# B&R Automation Studio project NAELD004C00R10L518F00 (part 50)

#### Act_Link.st
```iecst
(** 2018-12-08 **)
ACTION Act_Link:

	//Machine --> AGV ---> Communication On & Machine itself RUN Mode
	IF p_bLinkOpsRun = TRUE THEN

		tyDTMagToAGV.bCI4Auto := TRUE;
	ELSE
		tyDTMagToAGV.bCI4Auto	:= FALSE;
	END_IF

	tyDTMagToAGV.bCI4Occupied 			:= p_bBufferMagPresent OR p_bMagConvLftSen OR p_bMagConvRgtSen ;

	fbMagEmptyTm(IN:= p_bMagConvLftSen = FALSE AND p_bBufferMagPresent = FALSE);
	IF p_bBufferMagPresent AND p_tyLinkBufferStat.bBffrMty THEN
		tyDTMagToAGV.bCI4MagazineEmpty		:=  TRUE;
	ELSIF fbMagEmptyTm.Q THEN
		tyDTMagToAGV.bCI4MagazineEmpty		:=  FALSE;
	END_IF

	IF p_bLinkAGVOnline THEN

		p_tyAGVToDTMag.bVEHAuto		:= p_tyLinkAGVtoDTMag.bVEHAuto;
		p_tyAGVToDTMag.bVEHInPos1	:= p_tyLinkAGVtoDTMag.bVEHInPos1;
		p_tyAGVToDTMag.bVEHInPos2 	:= p_tyLinkAGVtoDTMag.bVEHInPos2;
		p_tyAGVToDTMag.bVEHInPos3 	:= p_tyLinkAGVtoDTMag.bVEHInPos3;
		p_tyAGVToDTMag.bVEHInPos4 	:= p_tyLinkAGVtoDTMag.bVEHInPos4 AND bAGVInPosSen;
		p_tyAGVToDTMag.bVEH1Occupied	:= p_tyLinkAGVtoDTMag.bVEH1Occupied;
		p_tyAGVToDTMag.bVEH2Occupied	:= p_tyLinkAGVtoDTMag.bVEH2Occupied;
		p_tyAGVToDTMag.bVEH3Occupied	:= p_tyLinkAGVtoDTMag.bVEH3Occupied;
		p_tyAGVToDTMag.bVEH4Occupied	:= p_tyLinkAGVtoDTMag.bVEH4Occupied;
		p_tyAGVToDTMag.bVEHRunning	:= p_tyLinkAGVtoDTMag.bVEHRunning;

	ELSE

		p_tyAGVToDTMag.bVEHAuto		:= FALSE;
		p_tyAGVToDTMag.bVEHInPos1	:= FALSE;
		p_tyAGVToDTMag.bVEHInPos2 	:= FALSE;
		p_tyAGVToDTMag.bVEHInPos3 	:= FALSE;
		p_tyAGVToDTMag.bVEHInPos4 	:= FALSE;
		p_tyAGVToDTMag.bVEH1Occupied:= FALSE;
		p_tyAGVToDTMag.bVEH2Occupied:= FALSE;
		p_tyAGVToDTMag.bVEH3Occupied:= FALSE;
		p_tyAGVToDTMag.bVEH4Occupied:= FALSE;
		p_tyAGVToDTMag.bVEHRunning	:= FALSE;

	END_IF

	bAIVInPos := p_tyAGVToDTMag.bVEHInPos4;
	bAIVAuto := p_tyAGVToDTMag.bVEHAuto;
	bAIVOccupied := p_tyAGVToDTMag.bVEH4Occupied;
	bMagConvAuto := tyDTMagToAGV.bCI4Auto;
	bMagConvOccupied :=  tyDTMagToAGV.bCI4Occupied;

	tyDTMagToAGV.bCI4Running := bMagConvRun;
	tyDTMagToAGV.bCI4Rdy	:= bMagConvRdy;

	IF p_bNtParamAGVInPosSenPrep THEN
		fbInPosErrTimer(IN:= p_tyLinkAGVtoDTMag.bVEHInPos3 AND bAGVInPosSen = FALSE, PT:= T#10s);
		IF fbInPosErrTimer.Q THEN
			eStatus		:= Error;
			udiStatus	:= 10009;	//AIV Not In Position
		END_IF
	END_IF

	IF p_bNtParamAGVInPosSenPrep THEN
		bAGVInPosSen := p_bAGVInPosSen1 AND p_bAGVInPosSen2;
	ELSE
		bAGVInPosSen := TRUE;
	END_IF

END_ACTION
```

#### Act_Main.st
```iecst
(** 2019-01-20 **)
ACTION Act_Main:

	IF eStatOld <> eStat THEN

		fbTxInTimer(IN := FALSE);
		fbTxOutTimer(IN := FALSE);
		fbMagOutTrig(CLK := FALSE);

		bMcRunRdy				 	  := FALSE;
		bRdyEnt			 		   	  := FALSE;
		bRdyExit				  	  := FALSE;
		bMagConvRun    := FALSE;
		fbCheckErrorTim(IN:= FALSE);
		usiStep		:= 0;

		sStatTxt	:= a_sStatText[eStat];

		eStatOld	:= eStat;

		eStatus		:= Busy;
	END_IF

	//Main
	CASE eStat OF

		AGVMagActIdle:
			eStatus	:= Idle;
			bMagConvRdy := FALSE;

		AGVMagActEnter:

			IF eStatus = Idle OR eStatus = Busy THEN

				eStatus	:= Busy;
				bMagConvRdy := TRUE;

				IF usiStep = 0 THEN

					IF bAIVAuto AND bMagConvAuto
						OR p_bSOTAvailable
						THEN // ON Connection

						bMagConvRdy  := TRUE; //Allow VEH to Move In

						IF bAIVInPos OR p_bSOTRcvOk THEN // VEH is in Position to Enter

							bRdyEnt := TRUE;

						END_IF
					END_IF

					IF bRdyEnt THEN

						IF bAIVInPos OR p_bSOTRcvOk  THEN

							bMagConvRdy := FALSE; // Temporarily Not Allowed Other VEH while one VEH in Pos.

							IF p_bSOTErr THEN
								eStatus		:= Error;
								udiStatus	:= 10010;//SOT Sensor Error Has Been Activated;

							ELSIF (NOT bMagConvOccupied) (*AND p_tyAGVToDTMag.bVEHOccupied*) THEN

								bMcRunRdy	:= TRUE;

								bMagConvRun := TRUE;

								usiStep	:= 1;
							ELSE
								eStatus		:= Error;
								udiStatus	:= 10000;	//Magazine Is Present Before Entering
							END_IF

						ELSE
							eStatus		:= Error;
							udiStatus	:= 10001;	//AIV Not In Enter Position
						END_IF

					END_IF

				ELSIF usiStep = 1 THEN

					IF p_eDirection = ConvDirLToL OR p_eDirection = ConvDirLToR THEN
						bEndSen	:= p_bMagConvRgtSen;
					ELSE
						bEndSen	:= p_bMagConvLftSen;
					END_IF

					fbTxInTimer(IN := TRUE, PT := DINT_TO_TIME(p_diTxInTimeOut));

					IF bEndSen = TRUE (*AND p_tyAGVToDTMag.bVEHOccupied = FALSE*) THEN

						eStatus	:= Done;

						bMagConvRdy := TRUE; // Allow VEH to Move Out After Transfering Magazine

						bMagConvRun := FALSE;

					ELSIF fbTxInTimer.Q = TRUE THEN

						eStatus		:= Error;
						udiStatus	:= 10002;	//Transfer In Time Out While Transporting

					END_IF

					IF bAIVInPos = FALSE AND p_bSOTRcvOk = FALSE AND eStatus = Busy THEN

						eStatus		:= Error;
						udiStatus	:= 10001;	//AIV Not In Enter Position
					END_IF

					//					IF bAIVAuto = FALSE AND eStatus = Busy THEN
					//
					//						eStatus		:= Error;
					//						udiStatus	:= 10006;	//AIV Not In Enter Position
					//					END_IF
				END_IF

			END_IF

		AGVMagActExit:
			IF eStatus = Idle OR eStatus = Busy THEN

				eStatus	:= Busy;

				bMagConvRdy := TRUE;

				IF usiStep = 0 THEN

					IF bAIVAuto AND bMagConvAuto
						OR p_bSOTRdy
						THEN // ON Connection

						bMagConvRdy  := TRUE; //Allow VEH to Move In

						IF bAIVInPos OR p_bSOTRcvOk THEN // VEH is in Position to Exit

							bRdyExit := TRUE;

						END_IF
					END_IF

					IF bRdyExit THEN

						IF (bAIVInPos OR p_bSOTRcvOk) AND bAIVOccupied=FALSE THEN

							bMagConvRdy := FALSE; // Temporarily Not Allowed Other VEH while one VEH in Pos.

							IF bMagConvOccupied OR p_bSOTRdy = FALSE THEN

								bMcRunRdy	:= TRUE;

								bMagConvRun := TRUE;

								usiStep	:= 1;

							ELSE
								eStatus		:= Error;
								udiStatus	:= 10003;	//Magazine Is Not Present Before Exiting
							END_IF

						ELSE
							eStatus		:= Error;
							udiStatus	:= 10004;	//AIV Not In Exit Position
						END_IF
					END_IF

				ELSIF usiStep = 1 THEN

					IF p_bSOTErr THEN

						usiStep := 2;
					END_IF

					IF p_eDirection = ConvDirLToR OR p_eDirection = ConvDirRToR THEN
						bEndSen	:= p_bMagConvRgtSen;
					ELSE
						bEndSen	:= p_bMagConvLftSen;
					END_IF

					fbTxOutTimer(IN := TRUE, PT := DINT_TO_TIME(p_diTxOutTimeOut));

					IF bEndSen = FALSE AND (bAIVOccupied = TRUE OR p_bSOTRdy = FALSE) THEN

						usiStep := 2;

					ELSIF fbTxOutTimer.Q = TRUE THEN

						eStatus		:= Error;
						udiStatus	:= 10005;	//Transfer Out Time Out While Transporting

					END_IF

					IF bAIVInPos = FALSE AND p_bSOTRcvOk = FALSE AND eStatus = Busy THEN

						eStatus		:= Error;
						udiStatus	:= 10001;	//AIV Not In Enter Position
					END_IF

					//					IF bAIVAuto = FALSE AND eStatus = Busy THEN
					//
					//						eStatus		:= Error;
					//						udiStatus	:= 10006;	//AIV Not In Auto
					//					END_IF

				ELSIF usiStep = 2 THEN
					fbCheckErrorTim(IN:= TRUE);
					IF p_bSOTErr THEN
						eStatus		:= Error;
						udiStatus	:= 10010;	//SOT Error signal activated
					ELSIF fbCheckErrorTim.Q THEN
						usiStep := 3;
					END_IF

				ELSIF usiStep = 3 THEN
					bMagConvRdy 	   := TRUE; // Allow VEH to Move Out After Transfering Magazine

					bMagConvRun := FALSE;
					eStatus := Done;
				END_IF

			END_IF
	END_CASE

END_ACTION
```

#### Init.st
```iecst
(** 2019-01-20 **)
PROGRAM _INIT

	(* Always Change If Project Change *)

	sProgNm	:= 'AGVMag 4';

	//Physical Configuration

	//Pass Address To Global Address For External Use
	//Action, State & Status
	p_AGVMag4Stat		:= ADR(eStat);
	p_AGVMag4Status		:= ADR(eStatus);
	p_AGVMag4StatTxt	:= ADR(sStatTxt);

	//Alarm
	p_AGVMag4AlmData	:= ADR(tyAlmData);

	//Output
	p_AGVMag4RdyEnter		:= ADR(bRdyEnt);
	p_AGVMag4RdyExit		:= ADR(bRdyExit);
	p_AGVMag4McRunRdy		:= ADR(bMcRunRdy);
	p_AGVMag4DTMagToAGV		:= ADR(tyDTMagToAGV);

	(* Always Change If Project Change *)

END_PROGRAM
```

### Program Logical/SOT/USSOT1 (IEC) - 1.00.0 - NtSOT v5.00.0

#### Act_InitGlobal.st
```iecst
(** 2021-04-20 **)
ACTION Act_InitGlobal:

	(* Always Change If Project Change *)

	//Pass Data To Link
	p_bLinkOpsRun ACCESS p_OpsRun;
	p_bLinkSOTReadyOnFirst ACCESS p_NtParamSOTReadyOnFirst;

	//Pass Data To Internal Use
	p_udiRstErr ACCESS p_RstErrReset;
	p_bManual ACCESS p_UIMnlMod;
	p_diTransferInTO ACCESS p_McParamMag1ConvRunTmOut;
	p_bEn ACCESS p_McParamAGVComEn;
//	p_bVirtualEn ACCESS p_UIVSOTUSEn;
//	p_bUBAVirtual ACCESS p_UIVSOTUBA;
	p_tRstDlyTm ACCESS p_NtParamUSSOT1RstDlyTm;
	p_tSigInChkTm ACCESS p_NtParamUSSOT1SigInChkTm;
	p_sProgNm ACCESS p_NtParamUSSOT1ProgNm;
	p_bNtSettingsLoadDone ACCESS p_StartupNtSettingsLoadDone;

	(* Always Change If Project Change *)

END_ACTION
```

#### Act_Link.st
```iecst
(** 2021-04-20 **)
ACTION Act_Link:

	//Ready Receive
	IF p_bLinkSOTReadyOnFirst THEN
		p_bRdyRcv	:= TRUE;
	ELSE
		p_bRdyRcv ACCESS p_DISOT1Available;
	END_IF

	p_bLeftSen ACCESS p_DIMagConvEntSen1;
	p_bRightSen ACCESS p_DIMagPresentSen1;
	p_bUMA ACCESS p_DISOT1Available;
	p_bUMASize ACCESS p_DISOT1SizeLarge;
	p_bDirLToR := TRUE;

	p_bComplSigOn	:= p_bRightSen;

END_ACTION
```

#### Act_LinkAction.st
```iecst
(** 2021-04-20 **)
ACTION Act_LinkAction:

	IF p_bLinkOpsRun = TRUE THEN
		p_eAct ACCESS p_OpsMagConvLD1USSOTAct;
	ELSE
		p_eAct ACCESS ADR(eAct);
	END_IF

END_ACTION
```

### Program Logical/SOT/DSSOT1 (IEC) - 1.00.0 - NtSOT v5.00.0

#### Act_InitGlobal.st
```iecst
(** 2021-04-20 **)
ACTION Act_InitGlobal:

	(* Always Change If Project Change *)

	//Pass Data To Link
	p_bLinkOpsRun ACCESS p_OpsRun;

	//Pass Data To Internal Use
	p_udiRstErr ACCESS p_RstErrReset;
	p_bManual ACCESS p_UIMnlMod;
	p_diTransferOutTO ACCESS p_McParamMag1ConvRunTmOut;
	p_bEn ACCESS p_McParamAGVComEn;
//	p_bVirtualEn ACCESS p_UIVSOTDSEn;
//	p_bDSBVirtual ACCESS p_UIVSOTDSB;
	p_tRstDlyTm ACCESS p_NtParamDSSOT1RstDlyTm;
	p_tSigInChkTm ACCESS p_NtParamDSSOT1SigInChkTm;
	p_sProgNm ACCESS p_NtParamDSSOT1ProgNm;
	p_bNtSettingsLoadDone ACCESS p_StartupNtSettingsLoadDone;

	p_bMagSizeLarge ACCESS p_OpsMagConvLD1MagSizeL;

	(* Always Change If Project Change *)

END_ACTION
```

#### Act_Link.st
```iecst
(** 2021-04-20 **)
ACTION Act_Link:

	//Ready Send
	p_bRdySend	:= TRUE;

	p_bLeftSen ACCESS p_DIMagConvEntSen1;
	p_bRightSen ACCESS p_DIMagPresentSen1;
	p_bDSB ACCESS p_DISOT1Ready;

	//Send Complete Signal
	IF EDGENEG(p_bLeftSen) THEN
		p_bComplSigOn	:= TRUE;
	END_IF

	IF eStat <> SOTActRun THEN
		p_bComplSigOn	:= FALSE;
	END_IF

END_ACTION
```

#### Act_LinkAction.st
```iecst
(** 2021-04-20 **)
ACTION Act_LinkAction:

	IF p_bLinkOpsRun = TRUE THEN
		p_eAct ACCESS p_OpsMagConvLD1DSSOTAct;
	ELSE
		p_eAct ACCESS ADR(eAct);
	END_IF

END_ACTION
```

### Program Logical/SOT/USSOT2 (IEC) - 1.00.0 - NtSOT v5.00.0

#### Act_Alarm.st
```iecst
(** 2021-04-20 **)
ACTION Act_Alarm:

	//Error
	IF EDGEPOS(eStatus = Error) THEN

		tyAlmData.sProgNm		:= p_sProgNm;
		tyAlmData.udiCode		:= udiStatus;
		tyAlmData.eSeverity		:= AlmSeverityError;
		tyAlmData.udiRunTime	:= tyAlmData.udiRunTime + 1;
		tyAlmData.bAlm			:= TRUE;
		tyAlmData.udiModuleNum  := udiModuleNum;
		g_sUSSOTProgNm		:= p_sProgNm;
		//Get Error Message
		IF tyAlmData.udiCode < 10000 OR tyAlmData.udiCode > 10099 THEN
			tyAlmData.sAlmMsg	:= 'Unknown';
			tyAlmData.sRcyMsg	:= 'Unknown';
		ELSE
			tyAlmData.sAlmMsg	:= a_tyAlmText[tyAlmData.udiCode].sAlmText;
			tyAlmData.sRcyMsg	:= a_tyAlmText[tyAlmData.udiCode].sRcyText;
		END_IF

		sStatTxt	:= tyAlmData.sAlmMsg;

	ELSIF bRstErr AND (tyAlmData.udiCode <> 0) THEN

		tyAlmData.udiCode	:= 0;
		tyAlmData.eSeverity	:= AlmSeverityNA;
		tyAlmData.sAlmMsg	:= '';
		tyAlmData.sRcyMsg	:= '';
		tyAlmData.bAlm			:= FALSE;
		sStatTxt	:= a_sStatText[eStat];

	END_IF

END_ACTION
```

#### Act_InitGlobal.st
```iecst
(** 2021-04-20 **)
ACTION Act_InitGlobal:

	(* Always Change If Project Change *)

	//Pass Data To Link
	p_bLinkOpsRun ACCESS p_OpsRun;
	p_bLinkSOTReadyOnFirst ACCESS p_NtParamSOTReadyOnFirst;

	//Pass Data To Internal Use
	p_udiRstErr ACCESS p_RstErrReset;
	p_bManual ACCESS p_UIMnlMod;
	p_diTransferInTO ACCESS p_McParamMag2ConvRunTmOut;
	p_bEn ACCESS p_McParamAGVComEn;
//	p_bVirtualEn ACCESS p_UIVSOTUSEn;
//	p_bUBAVirtual ACCESS p_UIVSOTUBA;
	p_tRstDlyTm ACCESS p_NtParamUSSOT2RstDlyTm;
	p_tSigInChkTm ACCESS p_NtParamUSSOT2SigInChkTm;
	p_sProgNm ACCESS p_NtParamUSSOT2ProgNm;
	p_bNtSettingsLoadDone ACCESS p_StartupNtSettingsLoadDone;

	(* Always Change If Project Change *)

END_ACTION
```

#### Act_Link.st
```iecst
(** 2021-04-20 **)
ACTION Act_Link:

	//Ready Receive
	IF p_bLinkSOTReadyOnFirst THEN
		p_bRdyRcv	:= TRUE;
	ELSE
		p_bRdyRcv ACCESS p_DISOT2Available;
	END_IF

	p_bLeftSen ACCESS p_DIMagConvEntSen2;
	p_bRightSen ACCESS p_DIMagPresentSen2;
	p_bUMA ACCESS p_DISOT2Available;
	p_bUMASize ACCESS p_DISOT2SizeLarge;
	p_bDirLToR := TRUE;

	p_bComplSigOn	:= p_bRightSen;

END_ACTION
```

#### Act_LinkAction.st
```iecst
(** 2021-04-20 **)
ACTION Act_LinkAction:

	IF p_bLinkOpsRun = TRUE THEN
		p_eAct ACCESS p_OpsMagConvLD2USSOTAct;
	ELSE
		p_eAct ACCESS ADR(eAct);
	END_IF

END_ACTION
```

### Program Logical/SOT/DSSOT2 (IEC) - 1.00.0 - NtSOT v5.00.0

#### Act_InitGlobal.st
```iecst
(** 2021-04-20 **)
ACTION Act_InitGlobal:

	(* Always Change If Project Change *)

	//Pass Data To Link
	p_bLinkOpsRun ACCESS p_OpsRun;

	//Pass Data To Internal Use
	p_udiRstErr ACCESS p_RstErrReset;
	p_bManual ACCESS p_UIMnlMod;
	p_diTransferOutTO ACCESS p_McParamMag2ConvRunTmOut;
	p_bEn ACCESS p_McParamAGVComEn;
//	p_bVirtualEn ACCESS p_UIVSOTDSEn;
//	p_bDSBVirtual ACCESS p_UIVSOTDSB;
	p_tRstDlyTm ACCESS p_NtParamDSSOT2RstDlyTm;
	p_tSigInChkTm ACCESS p_NtParamDSSOT2SigInChkTm;
	p_sProgNm ACCESS p_NtParamDSSOT2ProgNm;
	p_bNtSettingsLoadDone ACCESS p_StartupNtSettingsLoadDone;

	p_bMagSizeLarge ACCESS p_OpsMagConvLD2MagSizeL;

	(* Always Change If Project Change *)

END_ACTION
```

#### Act_Link.st
```iecst
(** 2021-04-20 **)
ACTION Act_Link:

	//Ready Send
	p_bRdySend	:= TRUE;

	p_bLeftSen ACCESS p_DIMagConvEntSen2;
	p_bRightSen ACCESS p_DIMagPresentSen2;
	p_bDSB ACCESS p_DISOT2Ready;

	//Send Complete Signal
	IF EDGENEG(p_bLeftSen) THEN
		p_bComplSigOn	:= TRUE;
	END_IF

	IF eStat <> SOTActRun THEN
		p_bComplSigOn	:= FALSE;
	END_IF

END_ACTION
```

#### Act_LinkAction.st
```iecst
(** 2021-04-20 **)
ACTION Act_LinkAction:

	IF p_bLinkOpsRun = TRUE THEN
		p_eAct ACCESS p_OpsMagConvLD2DSSOTAct;
	ELSE
		p_eAct ACCESS ADR(eAct);
	END_IF

END_ACTION
```

### USSOT3.var - Change By Project
```iecst
(*2021-03-19*)
(**)
(*Action & State & Status*)
VAR
	p_USSOT3Stat : UDINT;
	p_USSOT3Status : UDINT;
	p_USSOT3StatTxt : UDINT;
END_VAR
(**)
(*Alarm*)
VAR
	p_USSOT3AlmData : UDINT;
END_VAR
(**)
(*Output*)
VAR
	p_USSOT3USRdy : UDINT;
	p_USSOT3USLargeMagRdy : UDINT;
	p_USSOT3DSRdy : UDINT;
	p_USSOT3Transporting : UDINT;
	p_USSOT3ConvStart : UDINT;
	p_USSOT3ConvStop : UDINT;
	p_USSOT3USB : UDINT;
	p_USSOT3Virtual : UDINT;
END_VAR
```

### Program Logical/SOT/USSOT3 (IEC) - 1.00.0 - NtSOT v5.00.0

#### Act_InitGlobal.st
```iecst
(** 2021-04-20 **)
ACTION Act_InitGlobal:

	(* Always Change If Project Change *)

	//Pass Data To Link
	p_bLinkOpsRun ACCESS p_OpsRun;
	p_bLinkSOTReadyOnFirst ACCESS p_NtParamSOTReadyOnFirst;

	//Pass Data To Internal Use
	p_udiRstErr ACCESS p_RstErrReset;
	p_bManual ACCESS p_UIMnlMod;
	p_diTransferInTO ACCESS p_McParamMag3ConvRunTmOut;
	p_bEn ACCESS p_McParamAGVComEn;
//	p_bVirtualEn ACCESS p_UIVSOTUSEn;
//	p_bUBAVirtual ACCESS p_UIVSOTUBA;
	p_tRstDlyTm ACCESS p_NtParamUSSOT3RstDlyTm;
	p_tSigInChkTm ACCESS p_NtParamUSSOT3SigInChkTm;
	p_sProgNm ACCESS p_NtParamUSSOT3ProgNm;
	p_bNtSettingsLoadDone ACCESS p_StartupNtSettingsLoadDone;

	(* Always Change If Project Change *)

END_ACTION
```

#### Act_LinkAction.st
```iecst
(** 2021-04-20 **)
ACTION Act_LinkAction:

	IF p_bLinkOpsRun = TRUE THEN
		p_eAct ACCESS p_OpsMagConvLD3USSOTAct;
	ELSE
		p_eAct ACCESS ADR(eAct);
	END_IF

END_ACTION
```

### Program Logical/SOT/DSSOT3 (IEC) - 1.00.0 - NtSOT v5.00.0

#### Act_InitGlobal.st
```iecst
(** 2021-04-20 **)
ACTION Act_InitGlobal:

	(* Always Change If Project Change *)

	//Pass Data To Link
	p_bLinkOpsRun ACCESS p_OpsRun;

	//Pass Data To Internal Use
	p_udiRstErr ACCESS p_RstErrReset;
	p_bManual ACCESS p_UIMnlMod;
	p_diTransferOutTO ACCESS p_McParamMag3ConvRunTmOut;
	p_bEn ACCESS p_McParamAGVComEn;
//	p_bVirtualEn ACCESS p_UIVSOTDSEn;
//	p_bDSBVirtual ACCESS p_UIVSOTDSB;
	p_tRstDlyTm ACCESS p_NtParamDSSOT3RstDlyTm;
	p_tSigInChkTm ACCESS p_NtParamDSSOT3SigInChkTm;
	p_sProgNm ACCESS p_NtParamDSSOT3ProgNm;
	p_bNtSettingsLoadDone ACCESS p_StartupNtSettingsLoadDone;

	p_bMagSizeLarge ACCESS p_OpsMagConvLD3MagSizeL;

	(* Always Change If Project Change *)

END_ACTION
```

#### Act_LinkAction.st
```iecst
(** 2021-04-20 **)
ACTION Act_LinkAction:

	IF p_bLinkOpsRun = TRUE THEN
		p_eAct ACCESS p_OpsMagConvLD3DSSOTAct;
	ELSE
		p_eAct ACCESS ADR(eAct);
	END_IF

END_ACTION
```

### USSOT4.var - Change By Project
```iecst
(*2021-04-19*)
(**)
(*Action & State & Status*)
VAR
	p_USSOT4Stat : UDINT;
	p_USSOT4Status : UDINT;
	p_USSOT4StatTxt : UDINT;
END_VAR
(**)
(*Alarm*)
VAR
	p_USSOT4AlmData : UDINT;
END_VAR
(**)
(*Output*)
VAR
	p_USSOT4USRdy : UDINT;
	p_USSOT4USLargeMagRdy : UDINT;
	p_USSOT4DSRdy : UDINT;
	p_USSOT4Transporting : UDINT;
	p_USSOT4ConvStart : UDINT;
	p_USSOT4ConvStop : UDINT;
	p_USSOT4USB : UDINT;
	p_USSOT4Virtual : UDINT;
END_VAR
```

### Program Logical/SOT/USSOT4 (IEC) - 1.00.0 - NtSOT v5.00.0

#### InputRef_Link.var
```iecst
(*2021-04-20*)
(**)
VAR
	p_bLinkOpsRun : REFERENCE TO BOOL;
	p_bLinkSOTReadyOnFirst : REFERENCE TO BOOL;
END_VAR
```

#### Act_InitGlobal.st
```iecst
(** 2021-04-20 **)
ACTION Act_InitGlobal:

	(* Always Change If Project Change *)

	//Pass Data To Link
	p_bLinkOpsRun ACCESS p_OpsRun;
	p_bLinkSOTReadyOnFirst ACCESS p_NtParamSOTReadyOnFirst;

	//Pass Data To Internal Use
	p_udiRstErr ACCESS p_RstErrReset;
	p_bManual ACCESS p_UIMnlMod;
	p_diTransferInTO ACCESS p_McParamMag4ConvRunTmOut;
	p_bEn ACCESS p_McParamAGVComEn;
//	p_bVirtualEn ACCESS p_UIVSOTUSEn;
//	p_bUBAVirtual ACCESS p_UIVSOTUBA;
	p_tRstDlyTm ACCESS p_NtParamUSSOT4RstDlyTm;
	p_tSigInChkTm ACCESS p_NtParamUSSOT4SigInChkTm;
	p_sProgNm ACCESS p_NtParamUSSOT4ProgNm;
	p_bNtSettingsLoadDone ACCESS p_StartupNtSettingsLoadDone;

	(* Always Change If Project Change *)

END_ACTION
```

#### Act_Link.st
```iecst
(** 2021-04-20 **)
ACTION Act_Link:

	//Ready Receive
	IF p_bLinkSOTReadyOnFirst THEN
		p_bRdyRcv	:= TRUE;
	ELSE
		p_bRdyRcv ACCESS p_DISOT4Available;
	END_IF
	p_bLeftSen ACCESS p_DIMagConvEntSen4;
	p_bRightSen ACCESS p_DIMagPresentSen4;
	p_bUMA ACCESS p_DISOT4Available;
	p_bUMASize ACCESS p_DISOT4SizeLarge;
	p_bDirLToR := TRUE;

	p_bComplSigOn	:= p_bRightSen;

END_ACTION
```

#### Act_LinkAction.st
```iecst
(** 2021-04-20 **)
ACTION Act_LinkAction:

	IF p_bLinkOpsRun = TRUE THEN
		p_eAct ACCESS p_OpsMagConvLD4USSOTAct;
	ELSE
		p_eAct ACCESS ADR(eAct);
	END_IF

END_ACTION
```

#### Init.st
```iecst
(** 2021-04-20 **)
PROGRAM _INIT

	(* Always Change If Project Change *)

	//Pass Address To Global Address For External Use
	//Action, State & Status
	p_USSOT4Stat		:= ADR(eStat);
	p_USSOT4Status	:= ADR(eStatus);
	p_USSOT4StatTxt	:= ADR(sStatTxt);

	//Alarm
	p_USSOT4AlmData	:= ADR(tyAlmData);

	//Output
	p_USSOT4USRdy			:= ADR(bUSRdy);
	p_USSOT4USLargeMagRdy	:= ADR(bUSLargeMagRdy);
	p_USSOT4DSRdy			:= ADR(bDSRdy);
	p_USSOT4Transporting	:= ADR(bTransporting);
	p_USSOT4ConvStart		:= ADR(bConvStart);
	p_USSOT4ConvStop		:= ADR(bConvStop);
	p_USSOT4USB				:= ADR(bUSB);
	p_USSOT4Virtual			:= ADR(bVirtual);

	(* Always Change If Project Change *)

END_PROGRAM
```

### DSSOT4.var - Change By Project
```iecst
(*2021-04-20*)
(**)
(*Action & State & Status*)
VAR
	p_DSSOT4Stat : UDINT;
	p_DSSOT4Status : UDINT;
	p_DSSOT4StatTxt : UDINT;
END_VAR
(**)
(*Alarm*)
VAR
	p_DSSOT4AlmData : UDINT;
END_VAR
(**)
(*Output*)
VAR
	p_DSSOT4USRdy : UDINT;
	p_DSSOT4DSRdy : UDINT;
	p_DSSOT4Transporting : UDINT;
	p_DSSOT4ConvStart : UDINT;
	p_DSSOT4ConvStop : UDINT;
	p_DSSOT4DBA : UDINT;
	p_DSSOT4MagSizeLarge : UDINT;
	p_DSSOT4Virtual : UDINT;
END_VAR
```

### Program Logical/SOT/DSSOT4 (IEC) - 1.00.0 - NtSOT v5.00.0

#### Act_InitGlobal.st
```iecst
(** 2021-04-20 **)
ACTION Act_InitGlobal:

	(* Always Change If Project Change *)

	//Pass Data To Link
	p_bLinkOpsRun ACCESS p_OpsRun;

	//Pass Data To Internal Use
	p_udiRstErr ACCESS p_RstErrReset;
	p_bManual ACCESS p_UIMnlMod;
	p_diTransferOutTO ACCESS p_McParamMag4ConvRunTmOut;
	p_bEn ACCESS p_McParamAGVComEn;
//	p_bVirtualEn ACCESS p_UIVSOTDSEn;
//	p_bDSBVirtual ACCESS p_UIVSOTDSB;
	p_tRstDlyTm ACCESS p_NtParamDSSOT4RstDlyTm;
	p_tSigInChkTm ACCESS p_NtParamDSSOT4SigInChkTm;
	p_sProgNm ACCESS p_NtParamDSSOT4ProgNm;
	p_bNtSettingsLoadDone ACCESS p_StartupNtSettingsLoadDone;

	p_bMagSizeLarge ACCESS p_OpsMagConvLD4MagSizeL;

	(* Always Change If Project Change *)

END_ACTION
```

#### Act_Link.st
```iecst
(** 2021-04-20 **)
ACTION Act_Link:

	//Ready Send
	p_bRdySend	:= TRUE;

	p_bLeftSen ACCESS p_DIMagConvEntSen4;
	p_bRightSen ACCESS p_DIMagPresentSen4;
	p_bDSB ACCESS p_DISOT4Ready;

	//Send Complete Signal
	IF EDGENEG(p_bLeftSen) THEN
		p_bComplSigOn	:= TRUE;
	END_IF

	IF eStat <> SOTActRun THEN
		p_bComplSigOn	:= FALSE;
	END_IF

END_ACTION
```

#### Act_LinkAction.st
```iecst
(** 2021-04-20 **)
ACTION Act_LinkAction:

	IF p_bLinkOpsRun = TRUE THEN
		p_eAct ACCESS p_OpsMagConvLD4DSSOTAct;
	ELSE
		p_eAct ACCESS ADR(eAct);
	END_IF

END_ACTION
```

#### Init.st
```iecst
(** 2021-04-20 **)
PROGRAM _INIT

	(* Always Change If Project Change *)

	//Pass Address To Global Address For External Use
	//Action, State & Status
	p_DSSOT4Stat		:= ADR(eStat);
	p_DSSOT4Status		:= ADR(eStatus);
	p_DSSOT4StatTxt		:= ADR(sStatTxt);

	//Alarm
	p_DSSOT4AlmData	:= ADR(tyAlmData);

	//Output
	p_DSSOT4USRdy			:= ADR(bUSRdy);
	p_DSSOT4DSRdy			:= ADR(bDSRdy);
	p_DSSOT4Transporting	:= ADR(bTransporting);
	p_DSSOT4ConvStart		:= ADR(bConvStart);
	p_DSSOT4ConvStop		:= ADR(bConvStop);
	p_DSSOT4DBA				:= ADR(bDBA);
	p_DSSOT4Virtual			:= ADR(bVirtual);
	p_DSSOT4MagSizeLarge	:= ADR(bDSMagSizeLarge);

	(* Always Change If Project Change *)

END_PROGRAM
```

### Program Logical/Machine/Machine (IEC) - 1.00.0 - 

#### InputRef.var
```iecst
(*2019-03-22*)
(**)
(*General*)
VAR
	p_udiRstErr : REFERENCE TO UDINT;
END_VAR
(**)
(*Configuration*)
VAR
	p_bOpsRun : REFERENCE TO BOOL;
	p_bDIPressureSW : REFERENCE TO BOOL;
	p_diProdRcpCurrRcpWidth : REFERENCE TO DINT;
	p_diMagRcpCurrRcpMaxWidth : REFERENCE TO DINT;
	p_eStartupStep : REFERENCE TO eStartupStep;
END_VAR
(**)
VAR
	p_sProgNm : REFERENCE TO STRING[15];
	p_bNtSettingsLoadDone : REFERENCE TO BOOL;
	p_eLinkMag : REFERENCE TO eLDMag;
	p_usiLinkMod : REFERENCE TO USINT;
	p_bMcParamHermesSvyEn : REFERENCE TO BOOL;
END_VAR
```

#### Local.var
```iecst
(*2019-03-25*)
(**)
(*Local Action, State & Status*)
VAR
	eStatus : eFBStatus := Idle;
	udiStatus : UDINT := 0;
	udiStatus1 : UDINT := 0;
END_VAR
(**)
(*Local Alarm*)
VAR
	tyAlmData : tyAlmDat;
	tyAlmData1 : tyAlmDat;
	a_tyAlmText : ARRAY[10000..10099] OF tyAlmTxt := [(sAlmText:='Selected Product Width Exceeds Selected Magazine Maximum Board Width',sRcyText:='Please Reselect  Product or Magazine '),99(0)];
END_VAR
(**)
(*Local Output*)
(**)
(*Local Input*)
VAR
	udiRstErr : UDINT := 0;
END_VAR
(**)
VAR
	bOpsRun : BOOL;
	diProdRcpCurrRcpWidth : DINT;
	diMagRcpCurrRcpMaxWidth : DINT;
END_VAR
(**)
VAR
	sProgNm : STRING[15] := 'Machine';
	bNtSettingsLoadDone : BOOL := TRUE;
END_VAR
(**)
(*Local*)
VAR
	bRstErr : BOOL;
	udiRstErrOld : UDINT;
	bInitDone : BOOL;
	bInitialDone : BOOL;
END_VAR
(**)
VAR
	sBarcodeOut : STRING[255];
	bUSBDisconnected : BOOL;
	eStat : eUSBRdrAction := USBRdrActIdle;
	eMainStatus : eFBStatus := Idle;
	sStatTxt : STRING[200] := '';
	udiModuleNum : UDINT := 5951;
END_VAR
```

#### Act_Alarm.st
```iecst
(** 2019-03-25 **)
ACTION Act_Alarm:

	//Error
	IF EDGEPOS(eStatus = Error) THEN

		tyAlmData.sProgNm		:= p_sProgNm;
		tyAlmData.udiCode		:= udiStatus;
		tyAlmData.eSeverity		:= AlmSeverityError;
		tyAlmData.udiRunTime	:= tyAlmData.udiRunTime + 1;
		tyAlmData.bAlm			:= TRUE;
		tyAlmData.udiModuleNum  := udiModuleNum;
		g_sMachineProgNm		:= p_sProgNm;
		//Get Error Message
		IF tyAlmData.udiCode < 10000 OR tyAlmData.udiCode > 10099 THEN
			tyAlmData.sAlmMsg	:= 'Unknown';
			tyAlmData.sRcyMsg	:= 'Unknown';
		ELSE
			tyAlmData.sAlmMsg	:= a_tyAlmText[tyAlmData.udiCode].sAlmText;
			tyAlmData.sRcyMsg	:= a_tyAlmText[tyAlmData.udiCode].sRcyText;
		END_IF

	END_IF

END_ACTION
```

#### Act_Background.st
```iecst
(** 2019-01-23 **)
ACTION Act_Background:

	IF (p_diProdRcpCurrRcpWidth > p_diMagRcpCurrRcpMaxWidth) AND (eStatus <> Error) AND p_bMcParamHermesSvyEn =FALSE THEN

		eStatus		:= Error;
		udiStatus   := 10000;

	END_IF

	//Reset Error
	IF (eStatus = Error) AND bRstErr THEN
		eStatus		:= Idle;
		udiStatus	:= 0;
	END_IF

END_ACTION
```

#### Act_InitGlobal.st
```iecst
(** 2019-04-09 **)
ACTION Act_InitGlobal:

	(* Always Change If Project Change *)

	//Pass Data To Link
	p_eLinkMag ACCESS p_NtParamProjMag;
	p_usiLinkMod ACCESS p_ProdRcpCurrRcp0McMod;
	p_bMcParamHermesSvyEn ACCESS p_McParamHermesSvyEn;

	//Pass Data To Internal Use
	p_udiRstErr ACCESS p_RstErrReset;

	p_bOpsRun ACCESS p_OpsRun;
	p_eStartupStep ACCESS p_StartupStep;

	p_sProgNm ACCESS p_NtParamMcProgNm;
	p_bNtSettingsLoadDone ACCESS p_StartupNtSettingsLoadDone;

	(* Always Change If Project Change *)

END_ACTION
```

#### Act_Initial.st
```iecst
(** 2018-12-07 **)
ACTION Act_Initial:

	//Initial

END_ACTION
```

#### Act_Link.st
```iecst
(** 2018-12-11 **)
ACTION Act_Link:

	IF p_eLinkMag = LDMagQuadruple THEN
		CASE p_usiLinkMod OF
			0,2:
				p_diProdRcpCurrRcpWidth ACCESS p_ProdRcpCurrRcp0Width;
				p_diMagRcpCurrRcpMaxWidth ACCESS p_MagRcpCurrRcpMagMaxBrdWidth;

			1:
				p_diProdRcpCurrRcpWidth ACCESS p_ProdRcpCurrRcp0WidthRear;
				p_diMagRcpCurrRcpMaxWidth ACCESS p_MagRcpCurrRcpMagMaxBrdWidth1;
		END_CASE
	ELSE
		p_diProdRcpCurrRcpWidth ACCESS p_ProdRcpCurrRcp0Width;
		p_diMagRcpCurrRcpMaxWidth ACCESS p_MagRcpCurrRcpMagMaxBrdWidth;
	END_IF

END_ACTION
```

#### Init.st
```iecst
(** 2019-03-22 **)
PROGRAM _INIT

	(* Always Change If Project Change *)

	//Pass Address To Global Address For External Use
	//Action, State & Status

	//Alarm
	p_McAlmData		:= ADR(tyAlmData);
	p_McInfoData1	:= ADR(tyAlmData1);

	//Output

END_PROGRAM
```

### Machine1.var - Change By Project
```iecst
(*2018-12-07*)
(**)
(*Action & State & Status*)
(**)
(*Alarm*)
VAR
	p_Mc1AlmData : UDINT;
	p_Mc1InfoData1 : UDINT;
END_VAR
(**)
(*Output*)
```

### Program Logical/Machine/Machine1 (IEC, version 1.00.0) - 1.00.0 - 

#### Init.st - Change By Project
```iecst
(** 2019-03-22 **)
PROGRAM _INIT

	(* Always Change If Project Change *)

	//Pass Address To Global Address For External Use
	//Action, State & Status

	//Alarm
	p_Mc1AlmData		:= ADR(tyAlmData);
	p_Mc1InfoData1		:= ADR(tyAlmData1);

	//Output

	(* Always Change If Project Change *)

END_PROGRAM
```

#### Act_InitGlobal.st - Change By Project
```iecst
(** 2019-04-09 **)
ACTION Act_InitGlobal:

	(* Always Change If Project Change *)

	//Pass Data To Link
	p_eLinkMag ACCESS p_NtParamProjMag;
	p_usiLinkMod ACCESS p_ProdRcpCurrRcp0McMod;
	//Pass Data To Internal Use
	p_udiRstErr ACCESS p_RstErrReset;

	p_bOpsRun ACCESS p_OpsRun;
	p_eStartupStep ACCESS p_StartupStep;

	p_sProgNm ACCESS p_NtParamMc1ProgNm;
	p_bNtSettingsLoadDone ACCESS p_StartupNtSettingsLoadDone;

	(* Always Change If Project Change *)

END_ACTION
```

#### Act_Link.st - Change By Project
```iecst
(** 2018-12-11 **)
ACTION Act_Link:

	IF p_eLinkMag = LDMagQuadruple THEN
		CASE p_usiLinkMod OF
			1,2:
				p_diProdRcpCurrRcpWidth ACCESS p_ProdRcpCurrRcp0WidthRear;
				p_diMagRcpCurrRcpMaxWidth ACCESS p_MagRcpCurrRcpMagMaxBrdWidth1;

			0:
				p_diProdRcpCurrRcpWidth ACCESS p_ProdRcpCurrRcp0Width;
				p_diMagRcpCurrRcpMaxWidth ACCESS p_MagRcpCurrRcpMagMaxBrdWidth;
		END_CASE
	ELSE
		p_diProdRcpCurrRcpWidth := 0;
		p_diMagRcpCurrRcpMaxWidth := p_NtParamProdRcpMaxWidth;
	END_IF

END_ACTION
```

#### Cyclic.st - Change By Project
```iecst
(** 2019-03-22 **)
PROGRAM _CYCLIC

	IF bInitDone = FALSE THEN
		bInitDone	:= TRUE;

		Act_InitLocal;
		Act_InitGlobal;

	ELSIF bInitialDone = FALSE THEN

		//Special Case --> only after reading Current Recipe --> Excusively for Machine with Magazine Maximum Board Width Setting

		IF p_bNtSettingsLoadDone = TRUE AND p_eStartupStep = StartupStepUsrMgmt  THEN
			bInitialDone	:= TRUE;

			Act_Initial;
		END_IF

	ELSE

		Act_RstErr;
		Act_Link;
		Act_Background;
		Act_Alarm;
		Act_AlarmInfo1;

	END_IF

END_PROGRAM
```

#### Act_Alarm.st - Change By Project
```iecst
(** 2019-03-25 **)
ACTION Act_Alarm:

	//Error
	IF EDGEPOS(eStatus = Error) THEN

		tyAlmData.sProgNm		:= p_sProgNm;
		tyAlmData.udiCode		:= udiStatus;
		tyAlmData.eSeverity		:= AlmSeverityError;
		tyAlmData.udiRunTime	:= tyAlmData.udiRunTime + 1;
		tyAlmData.bAlm			:= TRUE;
		tyAlmData.udiModuleNum  := udiModuleNum;
		g_sMachineProgNm		:= p_sProgNm;
		//Get Error Message
		IF tyAlmData.udiCode < 10000 OR tyAlmData.udiCode > 10099 THEN
			tyAlmData.sAlmMsg	:= 'Unknown';
			tyAlmData.sRcyMsg	:= 'Unknown';
		ELSE
			tyAlmData.sAlmMsg	:= a_tyAlmText[tyAlmData.udiCode].sAlmText;
			tyAlmData.sRcyMsg	:= a_tyAlmText[tyAlmData.udiCode].sRcyText;
		END_IF

	END_IF

END_ACTION
```

#### InputRef.var - Change By Project
```iecst
(*2019-03-22*)
(**)
(*General*)
VAR
	p_udiRstErr : REFERENCE TO UDINT;
	p_bPrep : REFERENCE TO BOOL;
	p_bEn : REFERENCE TO BOOL;
	p_bDis : REFERENCE TO BOOL;
END_VAR
(**)
(*Configuration*)
VAR
	p_bOpsRun : REFERENCE TO BOOL;
	p_bDIPressureSW : REFERENCE TO BOOL;
	p_diProdRcpCurrRcpWidth : REFERENCE TO DINT;
	p_diMagRcpCurrRcpMaxWidth : REFERENCE TO DINT;
	p_eStartupStep : REFERENCE TO eStartupStep;
END_VAR
(**)
VAR
	p_sProgNm : REFERENCE TO STRING[15];
	p_bNtSettingsLoadDone : REFERENCE TO BOOL;
	p_eLinkMag : REFERENCE TO eLDMag;
	p_usiLinkMod : REFERENCE TO USINT;
END_VAR
```

#### Local.var - Change By Project
```iecst
(*2019-03-25*)
(**)
(*Local Action, State & Status*)
VAR
	eStatus : eFBStatus := Idle;
	udiStatus : UDINT := 0;
	udiStatus1 : UDINT := 0;
END_VAR
(**)
(*Local Alarm*)
VAR
	tyAlmData : tyAlmDat;
	tyAlmData1 : tyAlmDat;
	a_tyAlmText : ARRAY[10000..10099] OF tyAlmTxt := [(sAlmText:='Selected Product Width Exceeds Slected Magazine Maximum Board Width',sRcyText:='Please Reslect  Product or Magazine '),99((0))];
END_VAR
(**)
(*Local Output*)
(**)
(*Local Input*)
VAR
	udiRstErr : UDINT := 0;
END_VAR
(**)
VAR
	bOpsRun : BOOL;
	diProdRcpCurrRcpWidth : DINT;
	diMagRcpCurrRcpMaxWidth : DINT;
END_VAR
(**)
VAR
	sProgNm : STRING[15] := 'Machine';
	bNtSettingsLoadDone : BOOL := TRUE;
END_VAR
(**)
(*Local*)
VAR
	bRstErr : BOOL;
	udiRstErrOld : UDINT;
	bInitDone : BOOL;
	bInitialDone : BOOL;
	udiModuleNum : UDINT := 5951;
END_VAR
```

### BarcodeRdr.var - Change By Project
```iecst
(*2020-08-29 *)
(**)
(*Action & State & Status*)
VAR
	p_USBRdrStat : UDINT;
	p_USBRdrStatus : UDINT;
	p_USBRdrStatTxt : UDINT;
	p_USBudiStatus : UDINT;
END_VAR
(**)
(*Alarm*)
VAR
	p_USBRdrAlmData : UDINT;
	p_USBRdrAlmData1 : UDINT;
	p_USBRdrAlmData2 : UDINT;
END_VAR
(**)
(*Output*)
VAR
	p_USBDisconnected : UDINT;
	p_USBRdrBarcodeOut : UDINT;
END_VAR
```

### BarcodeRdr.typ - Change By Project
```iecst
(*2020-08-29*)
(**)
(*Action*)

TYPE
	eUSBRdrAction :
		(
		USBRdrActIdle,
		USBRdrActDetectDev,
		USBRdrActRead,
		USBRdrActSafetyRmv,
		USBRdrActFrmClose,
		USBRdrActCreateDir,
		USBRdrActDeleteOldLog
		);
END_TYPE

(**)
```

### Program Logical/USBBarcodeRdr/BarcodeRdr (IEC, version 1.00.1) - 1.00.1 - NtUSB v5.00.4 //
1.00.0 - Reading data from a barcode reader

#### Init.st - Change By Project
```iecst
(** 2020-08-29 **)
PROGRAM _INIT

	(* Always Change If Project Change *)

	//Pass Address To Global Address For External Use
	//Action, State & Status
	p_USBRdrStat		:= ADR(eStat);
	p_USBRdrStatus		:= ADR(eMainStatus);
	p_USBRdrStatTxt		:= ADR(sStatTxt);

	//Alarm
	p_USBRdrAlmData		:= ADR(tyAlmData);
	p_USBRdrAlmData1	:= ADR(tyAlmData1);
	p_USBRdrAlmData2	:= ADR(tyAlmData2);

	//Output
	p_USBRdrBarcodeOut 	:= ADR(sBarcodeOut);
	p_USBDisconnected   := ADR(bUSBDisconnected);
	(* Always Change If Project Change *)

END_PROGRAM
```

#### Act_InitGlobal.st - Change By Project
```iecst
(** 2020-08-29 **)
ACTION Act_InitGlobal:

	(* Always Change If Project Change *)

	//Pass Data To Link
	p_bLinkOpsRun ACCESS p_OpsRun;
	p_bLinkStartupRun ACCESS p_StartupRun;
	p_tyLinkNtParam ACCESS p_NtParamCurr;

	//Pass Data To Internal Use
	p_udiRstErr ACCESS p_RstErrReset;
	p_bManual ACCESS p_UIMnlMod;
	p_sProgNm ACCESS p_NtParamUSBProgNm;

    p_eAct ACCESS p_UIUSBRdrAct;       //ADD

	p_diVendorID ACCESS p_McParamVID;
	p_diProductID ACCESS p_McParamPID;
	p_bUSBRun ACCESS p_UIUSBRun;
	p_bScannerEn ACCESS p_McParamScannerEn;

	p_dtCurrDT ACCESS p_TimeCurrDT;
	p_udiFileKeepDay ACCESS p_NtParamAlmFileKeepDay;
	p_bNtSettingsLoadDone ACCESS p_StartupNtSettingsLoadDone;

	(* Always Change If Project Change *)

END_ACTION
```

#### InputRef_Link.var - Change By Project
```iecst
(*2020-08-29*)
(**)
VAR
	p_bLinkOpsRun : REFERENCE TO BOOL;
	p_tyLinkNtParam : REFERENCE TO tyNtParam;
	p_bLinkStartupRun : REFERENCE TO BOOL;
END_VAR
```

#### Act_LinkAction.st - Change By Project
```iecst
(** 2020-08-29 **)
ACTION Act_LinkAction:

	IF p_bLinkStartupRun = TRUE THEN
		p_eAct ACCESS p_StartupUSBAct;
	ELSE
		p_eAct ACCESS p_UIUSBRdrAct;
	END_IF

END_ACTION
```

#### Act_LinkEn.st - Change By Project
```iecst
(** 2020-08-29 **)
ACTION Act_LinkEn:

	//Link bPrep, bEn & bDis
//	p_bPrep := (p_tyLinkNtParam.bBCodeScannerPrep) AND (p_tyLinkNtParam.eScannerType = USB);
	p_bEn 	:= p_tyLinkNtParam.bUSBScannerPrep;
END_ACTION
```

#### Act_Link.st - Change By Project
```iecst
(** 2020-08-29 **)
ACTION Act_Link:

END_ACTION
```

#### Act_Initial.st - Do Not Change!!!
```iecst
(** 2020-08-29 **)
ACTION Act_Initial:

	//Initial
	sStatTxt	:= a_sStatText[eStat];

	fbGetUSBDevice.uiFilterInterfaceClass := 3; // HID
	fbGetUSBDevice.uiFilterInterfaceSubClass := 1; //HID
	fbGetUSBDevice (bEn := FALSE);
	fbReadUSBDevice (bEn := FALSE);
	fbRmvUSBDevice (bEn := FALSE);

	fbDirCreate1.sDevice	:= 'F';
	fbDirCreate1.sDirName	:= 'User';
	fbDirCreate1(bEn := FALSE);

	fbDirCreate2.sDevice	:= 'User';
	fbDirCreate2.sDirName	:= 'Serial';
	fbDirCreate2(bEn := FALSE);

	fbDirCreate3.sDevice	:= 'Serial';
	fbDirCreate3.sDirName	:= 'USB';
	fbDirCreate3(bEn := FALSE);

	fbFileAppend1.sDevice	:= 'USB';
	fbFileAppend1(bEn := FALSE);

	fbFileOldDel1.sDevice	:= 'USB';
	fbFileOldDel1.sPath		:= '';
	fbFileOldDel1.sKeyword	:= 'USB_';
	fbFileOldDel1(bEn := FALSE);

END_ACTION
```

#### Cyclic.st - Do Not Change!!!
```iecst
(** 2020-08-29 **)
PROGRAM _CYCLIC

	IF bInitDone = FALSE THEN
		bInitDone	:= TRUE;

		Act_InitLocal;
		Act_InitGlobal;

	ELSIF bInitialDone = FALSE  THEN
		IF p_bNtSettingsLoadDone = TRUE THEN
			bInitialDone	:= TRUE;

			Act_Initial;
		END_IF

	ELSE

		Act_RstErr;
		Act_LinkAction;
		Act_Action;
		Act_LinkEn;

		IF (p_bPrep = TRUE) AND (p_bEn = TRUE) AND (p_bDis = FALSE) THEN
			Act_Link;
			Act_Main;
			Act_Background;
		ELSE
			IF eStat <> USBRdrActIdle THEN
				eStatus	:= Done;
			ELSE
				eStatus	:= Idle;
			END_IF
		END_IF

		Act_CombineErr;
		Act_Alarm;
		Act_Alarm1;
		Act_Alarm2;

	END_IF

END_PROGRAM
```

#### Act_RstErr.st - Do Not Change!!!
```iecst
(** 2020-08-29 **)
ACTION Act_RstErr:

	IF p_udiRstErr <> udiRstErrOld THEN
		bRstErr			:= TRUE;
		udiRstErrOld	:= p_udiRstErr;
	ELSE
		bRstErr			:= FALSE;
	END_IF

END_ACTION
```

#### Act_Action.st - Do Not Change!!!
```iecst
(** 2020-08-29 **)
ACTION Act_Action:

		//Reset Error
	IF (eStatus = Error) AND bRstErr THEN
		p_eAct	:= USBRdrActIdle;
		eStat	:= USBRdrActIdle;
	END_IF

	//Set p_eAct
	IF eStatus = Idle OR eStatus = Busy OR eStatus = Done THEN
		eStat	:= p_eAct;
	END_IF

	IF eStatus = Error THEN
		fbRmvUSBDevice (bEn := TRUE, udiUSBIdent := fbReadUSBDevice.udiUSBIdent );
		IF fbRmvUSBDevice.udiStatus = 0 THEN
			fbRmvUSBDevice(bEn := FALSE);
			p_eAct	:= USBRdrActIdle;
		ELSIF fbRmvUSBDevice.udiStatus < 65534 THEN
			fbRmvUSBDevice(bEn := FALSE);
			p_eAct	:= USBRdrActIdle;
		END_IF
	END_IF

END_ACTION
```

#### Act_InitLocal.st - Do Not Change!!!
```iecst
(** 2020-08-29 **)
ACTION Act_InitLocal:

	//Input Reference Link To Local Variable
	p_eAct ACCESS ADR(eAct);
	p_udiRstErr ACCESS ADR(udiRstErr);
	p_bPrep ACCESS ADR(bPrep);
	p_bEn ACCESS ADR(bEn);
	p_bDis ACCESS ADR(bDis);

	p_bManual ACCESS ADR(bManual);
	p_sProgNm ACCESS ADR(sProgNm);

	p_diVendorID ACCESS ADR (uiVendorID);
	p_diProductID ACCESS ADR (uiProductID);
	p_bUSBRun ACCESS ADR (bUSBRun);
	p_bScannerEn ACCESS ADR (bScannerEn);
	p_dtCurrDT ACCESS ADR(dtCurrDT);
	p_udiFileKeepDay ACCESS ADR(udiFileKeepDay);

	p_bNtSettingsLoadDone ACCESS ADR(bNtSettingsLoadDone);

END_ACTION
```

#### Act_Main.st - Do Not Change!!!
```iecst
(** 2020-12-29 **)
ACTION Act_Main:

	CASE eStat OF

		USBRdrActIdle:

			(*fbRmvUSBDevice 	(bEn := FALSE);*)
			sStatTxt	:= a_sStatText[eStat];
			eStatus	:= Idle;

			sBarcodeOut:= '';
			fbUSBTimer(IN := FALSE);
			bUSBDisconnected := FALSE;
			usiStep := 0;

			fbGetUSBDevice (bEn := FALSE);
			fbReadUSBDevice (bEn := FALSE);
			fbRmvUSBDevice (bEn := FALSE);
			fbDirCreate1(bEn := FALSE);
			fbDirCreate2(bEn := FALSE);
			fbDirCreate3(bEn := FALSE);

		USBRdrActDetectDev:

			IF eStatus = Idle OR eStatus = Busy THEN

				eStatus	:= Busy;
				CASE usiStep OF
					0:
						fbGetUSBDevice.uiVendorID 	:= DINT_TO_UINT (p_diVendorID);
						fbGetUSBDevice.uiProductID	:= DINT_TO_UINT (p_diProductID);
						fbGetUSBDevice (bEn := TRUE);

						fbUSBTimer(IN := TRUE);

						IF fbGetUSBDevice.udiStatus = 0 THEN
							eStatus := Done;
							bNodeExist := UDINT_TO_BOOL (fbGetUSBDevice.udiNodeId);
							fbUSBTimer(IN := FALSE);

							bUSBDisconnected := FALSE;

						ELSIF fbUSBTimer.Q = TRUE  THEN

							bUSBDisconnected := TRUE;

							udiStatus2 	:= 10004;
							usiStep := 99;
							fbUSBTimer(IN := FALSE);
						END_IF

					99:
						fbGetUSBDevice (bEn := FALSE);
				END_CASE
			END_IF

		USBRdrActRead:

			IF eStatus = Idle OR eStatus = Busy THEN

				eStatus	:= Busy;

				fbReadUSBDevice (bEn := TRUE, udiDevice := ADR(fbGetUSBDevice.asDeviceNm));
				bUSBRmv := FALSE;
				bNodeExist := UDINT_TO_BOOL (fbGetUSBDevice.udiNodeId);

				IF fbReadUSBDevice.udiStatus = 0 THEN

					eStatus	    := Done;

					sBarcodeOut := fbReadUSBDevice.sBarcodeOut;

					fbReadUSBDevice (bEn := FALSE);

					IF fbReadUSBDevice.bNewBarcode THEN //Record new barcode in log file
						fLogDTConvert(ADR(sDT) , p_dtCurrDT);
						memset(ADR(a_sLogList[udiLogCntr]) , 0 , SIZEOF(a_sLogList[udiLogCntr]));
						memcpy(ADR(a_sLogList[udiLogCntr]) + LEN(a_sLogList[udiLogCntr]) , ADR(sDT) , LEN(sDT));
						memcpy(ADR(a_sLogList[udiLogCntr]) + LEN(a_sLogList[udiLogCntr]) , ADR('$r$n') , LEN('$r$n'));
						memcpy(ADR(a_sLogList[udiLogCntr]) + LEN(a_sLogList[udiLogCntr]) , ADR('Received :') , LEN('Received :'));
						memcpy(ADR(a_sLogList[udiLogCntr]) + LEN(a_sLogList[udiLogCntr]) , ADR(sBarcodeOut) , LEN(sBarcodeOut));
						memcpy(ADR(a_sLogList[udiLogCntr]) + LEN(a_sLogList[udiLogCntr]) , ADR('$r$n$r$n') , LEN('$r$n$r$n'));

						udiLogCntr	:= udiLogCntr + 1;
						IF udiLogCntr = 10 THEN
							udiLogCntr	:= 0;
						END_IF
					END_IF

				ELSIF fbReadUSBDevice.udiStatus < 65534 THEN

					eStatus := Error;

					IF fbReadUSBDevice.udiStatus = 9667 THEN
						udiStatus 	:= 10000; //Device Lost Connection.

					ELSIF fbReadUSBDevice.udiStatus = 9668 THEN
						udiStatus 		:= 10002; //Device Not Found.
					ELSE
						udiStatus 		:= fbReadUSBDevice.udiStatus;
					END_IF

				END_IF

			END_IF

		USBRdrActSafetyRmv:
			IF eStatus = Idle OR eStatus = Busy THEN

				eStatus	:= Busy;

				sBarcodeOut := '';

				IF bUSBRmv = FALSE THEN
					fbRmvUSBDevice (bEn := TRUE, udiUSBIdent := fbReadUSBDevice.udiUSBIdent );

					IF fbRmvUSBDevice.udiStatus = 0 THEN
						eStatus := Done;
						bUSBRmv := TRUE;
						fbReadUSBDevice (bEn := FALSE);
						fbGetUSBDevice 	(bEn := FALSE);
						bNodeExist := UDINT_TO_BOOL (fbGetUSBDevice.udiNodeId);

					ELSIF fbRmvUSBDevice.udiStatus < 65534 THEN
						eStatus := Error;
						IF fbRmvUSBDevice.udiStatus = 8251 THEN
							udiStatus := 10003;
						END_IF

					END_IF
				END_IF
			END_IF

		USBRdrActFrmClose:
			IF eStatus = Idle OR eStatus = Busy THEN

				eStatus	:= Busy;
				fbRmvUSBDevice (bEn := TRUE, udiUSBIdent := fbReadUSBDevice.udiUSBIdent );

				sBarcodeOut := '';

				IF fbRmvUSBDevice.udiStatus = 0 THEN
					eStatus := Done;
					fbReadUSBDevice (bEn := FALSE);

				ELSIF fbRmvUSBDevice.udiStatus < 65534 THEN
					eStatus := Error;
					IF fbRmvUSBDevice.udiStatus = 8251 THEN
						udiStatus := 10003; //Device No Open.
					END_IF

				END_IF
			END_IF

		//Log file handling ----------------------------------------------
		USBRdrActCreateDir:
			IF eStatus = Idle OR eStatus = Busy THEN

				eStatus	:= Busy;

				sStatTxt	:= a_sStatText[eStat];

				CASE usiStep OF
					0:
						fbDirCreate1(bEn := TRUE);
						IF fbDirCreate1.udiStatus = 0 THEN
							usiStep	:= 1;
						ELSIF fbDirCreate1.udiStatus < 65534 THEN
							eStatus		:= Error;

							IF fbDirCreate1.udiStatus = 1908 THEN
								udiStatus	:= 10011;	//Create User Directory Error
							ELSE
								udiStatus	:= fbDirCreate1.udiStatus;
							END_IF
						END_IF

					1:
						fbDirCreate2(bEn := TRUE);
						IF fbDirCreate2.udiStatus = 0 THEN
							usiStep	:= 2;
						ELSIF fbDirCreate2.udiStatus < 65534 THEN
							eStatus		:= Error;

							IF fbDirCreate2.udiStatus = 1908 THEN
								udiStatus	:= 10012;	//Create Serial Directory Error
							ELSE
								udiStatus	:= fbDirCreate2.udiStatus;
							END_IF
						END_IF
					2:
						fbDirCreate3(bEn := TRUE);
						IF fbDirCreate3.udiStatus = 0 THEN
							eStatus	:= Done;
						ELSIF fbDirCreate3.udiStatus < 65534 THEN
							eStatus		:= Error;

							IF fbDirCreate3.udiStatus = 1908 THEN
								udiStatus	:= 10013;	//Create USB Directory Error
							ELSE
								udiStatus	:= fbDirCreate3.udiStatus;
							END_IF
						END_IF

				END_CASE

			END_IF

		USBRdrActDeleteOldLog:
			IF eStatus = Idle OR eStatus = Busy THEN

				eStatus	:= Busy;

				sStatTxt	:= a_sStatText[eStat];

				fbFileOldDel1.dtDTNow			:= p_dtCurrDT;
				fbFileOldDel1.udiFileKeepDay	:= p_udiFileKeepDay;
				fbFileOldDel1(bEn := TRUE);
				IF fbFileOldDel1.udiStatus = 0 THEN
					eStatus	:= Done;
				ELSIF fbFileOldDel1.udiStatus < 65534 THEN
					eStatus		:= Error;

					IF fbFileOldDel1.udiStatus = 1910 THEN
						udiStatus	:= 10014;	//Get Directory Info Error While Deleting Old Log
					ELSIF fbFileOldDel1.udiStatus = 1911 THEN
						udiStatus	:= 10015;	//Directory Read Error While Deleting Old Log
					ELSIF fbFileOldDel1.udiStatus = 1912 THEN
						udiStatus	:= 10016;	//File Delete Error While Deleting Old Log
					ELSE
						udiStatus	:= fbFileOldDel1.udiStatus;
					END_IF
				END_IF

			END_IF
	END_CASE

END_ACTION
```

#### Act_Background.st - Do Not Change!!!
```iecst
(** 2020-08-29 **)
ACTION Act_Background:

	IF (eStatus1 = Error) AND bRstErr THEN
		eStatus1	:= Idle;
		udiStatus1	:= 0;

		fbFileAppend1(bEn := FALSE);
		iWriteLogStep	:= 0;
	END_IF

	IF eStatus1 <> Error THEN

		IF udiWriteLogCntr <> udiLogCntr THEN

			CASE iWriteLogStep OF

				0:
					dtCurrDTTemp			:= p_dtCurrDT;
					fbFileAppend1.sFile		:= DT_TO_STRING(dtCurrDTTemp);
					fbFileAppend1.sFile		:= MID(fbFileAppend1.sFile , 10 , 4);
					fbFileAppend1.sFile		:= CONCAT('_' , fbFileAppend1.sFile);
					fbFileAppend1.sFile		:= CONCAT('USB' , fbFileAppend1.sFile);
					fbFileAppend1.sFile		:= CONCAT(fbFileAppend1.sFile , '.dat');

					fbFileAppend1.p_Src		:= ADR(a_sLogList[udiWriteLogCntr]);
					fbFileAppend1.udiLen	:= LEN(a_sLogList[udiWriteLogCntr]);

					iWriteLogStep	:= 1;

				1:
					fbFileAppend1(bEn := TRUE);
					IF fbFileAppend1.udiStatus = 0 THEN
						fbFileAppend1(bEn := FALSE);

						udiWriteLogCntr	:= udiWriteLogCntr + 1;
						IF udiWriteLogCntr = 10 THEN
							udiWriteLogCntr	:= 0;
						END_IF

						iWriteLogStep	:= 0;

					ELSIF fbFileAppend1.udiStatus < 65534 THEN
						eStatus1	:= Error;

						IF fbFileAppend1.udiStatus = 1900 THEN
							udiStatus1	:= 10017;	//File Open Error While Writing Serial Log
						ELSIF fbFileAppend1.udiStatus = 1901 THEN
							udiStatus1	:= 10018;	//File Create Error While Writing Serial Log
						ELSIF fbFileAppend1.udiStatus = 1913 THEN
							udiStatus1	:= 10019;	//Get File Info Error While Writing Serial Log
						ELSIF fbFileAppend1.udiStatus = 1903 THEN
							udiStatus1	:= 10020;	//File Write Error While Writing Serial Log
						ELSIF fbFileAppend1.udiStatus = 1904 THEN
							udiStatus1	:= 10021;	//File Close Error While Writing Serial Log
						ELSIF fbFileAppend1.udiStatus = 1914 THEN
							udiStatus1	:= 10022;	//Directory Does Not Exist While Writing Serial Log
						ELSE
							udiStatus1	:= fbFileAppend1.udiStatus;
						END_IF

						iWriteLogStep	:= 0;

					END_IF

			END_CASE

		END_IF

	END_IF
END_ACTION
```

#### Act_Alarm.st - Do Not Change!!!
```iecst
(** 2020-08-29 **)
ACTION Act_Alarm:

	//Error
	IF EDGEPOS(eStatus = Error) THEN

		tyAlmData.sProgNm		:= p_sProgNm;
		tyAlmData.udiCode		:= udiStatus;
		tyAlmData.eSeverity		:= AlmSeverityError;
		tyAlmData.udiRunTime	:= tyAlmData.udiRunTime + 1;
		tyAlmData.bAlm			:= TRUE;
		tyAlmData.udiModuleNum  := udiModuleNum;
		g_sBarcodeRdrProgNm		:= p_sProgNm;

		//Get Error Message
		IF tyAlmData.udiCode < 10000 OR tyAlmData.udiCode > 10199 THEN
			tyAlmData.sAlmMsg	:= 'Unknown';
			tyAlmData.sRcyMsg	:= 'Unknown';
		ELSE
			tyAlmData.sAlmMsg	:= a_tyAlmText[tyAlmData.udiCode].sAlmText;
			tyAlmData.sRcyMsg	:= a_tyAlmText[tyAlmData.udiCode].sRcyText;
		END_IF

		sStatTxt	:= tyAlmData.sAlmMsg;

	ELSIF bRstErr AND (tyAlmData.udiCode <> 0) THEN

		tyAlmData.udiCode	:= 0;
		tyAlmData.eSeverity	:= AlmSeverityNA;
		tyAlmData.sAlmMsg	:= '';
		tyAlmData.sRcyMsg	:= '';
		tyAlmData.bAlm			:= FALSE;
		sStatTxt	:= a_sStatText[eStat];

	END_IF

END_ACTION
```

#### Act_Alarm1.st - Do Not Change!!!
```iecst
(** 2020-08-29 **)
ACTION Act_Alarm1:

	//Error
	IF EDGEPOS(eStatus1 = Error) THEN

		tyAlmData1.sProgNm		:= p_sProgNm;
		tyAlmData1.udiCode		:= udiStatus1;
		tyAlmData1.eSeverity	:= AlmSeverityError;
		tyAlmData1.udiRunTime	:= tyAlmData1.udiRunTime + 1;
		tyAlmData1.bAlm			:= TRUE;
		tyAlmData1.udiModuleNum  := udiModuleNum;
		g_sBarcodeRdrProgNm		:= p_sProgNm;
		//Get Error Message
		IF tyAlmData1.udiCode < 10000 OR tyAlmData1.udiCode > 10199 THEN
			tyAlmData1.sAlmMsg	:= 'Unknown';
			tyAlmData1.sRcyMsg	:= 'Unknown';
		ELSE
			tyAlmData1.sAlmMsg	:= a_tyAlmText[tyAlmData1.udiCode].sAlmText;
			tyAlmData1.sRcyMsg	:= a_tyAlmText[tyAlmData1.udiCode].sRcyText;
		END_IF

		sStatTxt	:= tyAlmData1.sAlmMsg;

	ELSIF bRstErr AND (tyAlmData1.udiCode <> 0) THEN

		tyAlmData1.udiCode	:= 0;
		tyAlmData1.eSeverity	:= AlmSeverityNA;
		tyAlmData1.sAlmMsg	:= '';
		tyAlmData1.sRcyMsg	:= '';
		tyAlmData1.bAlm			:= FALSE;
		sStatTxt	:= a_sStatText[eStat];

	END_IF

END_ACTION
```

#### Act_Alarm2.st - Do Not Change!!!
```iecst
(** 2020-08-29 **)
ACTION Act_Alarm2:

	//Error
	IF  (eStatus<>Error) AND bUSBDisconnected AND p_bUSBRun AND p_bScannerEn = TRUE THEN

		tyAlmData2.sProgNm		:= p_sProgNm;
		tyAlmData2.udiCode		:= udiStatus2;
		tyAlmData2.eSeverity	:= AlmSeverityWarning;
		tyAlmData2.udiRunTime	:= tyAlmData2.udiRunTime + 1;
		tyAlmData2.bAlm			:= TRUE;
		tyAlmData2.udiModuleNum  := udiModuleNum;
		g_sBarcodeRdrProgNm		:= p_sProgNm;
		//Get Error Message
		IF tyAlmData2.udiCode < 10000 OR tyAlmData2.udiCode > 10199 THEN
			tyAlmData2.sAlmMsg	:= 'Unknown';
			tyAlmData2.sRcyMsg	:= 'Unknown';
		ELSE
			tyAlmData2.sAlmMsg	:= a_tyAlmText[tyAlmData2.udiCode].sAlmText;
			tyAlmData2.sRcyMsg	:= a_tyAlmText[tyAlmData2.udiCode].sRcyText;
		END_IF

		sStatTxt	:= tyAlmData2.sAlmMsg;

	ELSE

		tyAlmData2.udiCode	:= 0;
		tyAlmData2.eSeverity	:= AlmSeverityNA;
		tyAlmData2.sAlmMsg	:= '';
		tyAlmData2.sRcyMsg	:= '';
		tyAlmData2.bAlm			:= FALSE;
		sStatTxt	:= a_sStatText[eStat];

	END_IF

END_ACTION
```

#### InputRef.var - Do Not Change!!!
```iecst
(*2020-08-29*)
(**)
(*General*)
VAR
	p_eAct : REFERENCE TO eUSBRdrAction;
	p_udiRstErr : REFERENCE TO UDINT;
	p_bPrep : REFERENCE TO BOOL;
	p_bEn : REFERENCE TO BOOL;
	p_bDis : REFERENCE TO BOOL;
END_VAR
(**)
(*Configuration*)
VAR
	p_bManual : REFERENCE TO BOOL;
	p_sProgNm : REFERENCE TO STRING[15];
	p_bNtSettingsLoadDone : REFERENCE TO BOOL;
	p_dtCurrDT : REFERENCE TO DATE_AND_TIME;
	p_udiFileKeepDay : REFERENCE TO UDINT;
END_VAR
(**)
(*Input*)
VAR
	p_diVendorID : REFERENCE TO DINT;
	p_diProductID : REFERENCE TO DINT;
	p_bUSBRun : REFERENCE TO BOOL;
	p_bScannerEn : REFERENCE TO BOOL;
END_VAR
```

#### Local.var - Do Not Change!!!
```iecst
(* 2020-08-29 *)
(**)
(*Local Action, State & Status*)
VAR
	eAct : eUSBRdrAction := USBRdrActIdle;
	eStat : eUSBRdrAction := USBRdrActIdle;
	eMainStatus : eFBStatus := Idle;
	eStatus : eFBStatus := Idle;
	eStatus1 : eFBStatus := Idle;
	udiStatus : UDINT := 0;
	udiStatus1 : UDINT := 0;
	udiStatus2 : UDINT := 0;
	sStatTxt : STRING[200] := '';
	a_sStatText : ARRAY[0..60] OF STRING[200] := ['Idling','Initializing','Initializing With Reverse','Initializing With Pusher','Initializing With Puller','Initializing With Reject','Initializing With Inspection','Entering Board','Entering Board Until Inlet Signal Off','Entering Board With Reverse','Reversing Board','Reversing Board With Immediate Start Conv','Entering Board With Puller','Entering Board With Reject','Entering Board With Inspection','Pre Exiting Board','Resuming Reject Board',2('Exiting Board'),2('Exiting Board With Pusher'),'Pusher Setting All Control','Pusher Resetting All Control','Pusher Setting Extend','Pusher Setting Retract','Pusher Extending','Pusher Retracting','Puller Setting All Control','Puller Resetting All Control','Puller Setting Extend','Puller Setting Retract','Puller Extending','Puller Retracting','Rotating Setting All Control','Rotating Resetting All Control','Rotating Setting Home','Rotating Setting Remote','Rotating Turning Home','Rotating Turning Remote','Reject Setting All Control','Reject Resetting All Control','Reject Setting Up','Reject Setting Down','Reject Going Up','Reject Going Down','Stopping','Stopping With Pusher','Stopping With Puller','Stopping With Reject','Turning On Motor Signal','Turning On Motor Direction','Turning Off Motor Signal','Turning Off Motor Direction','Turning On All Motor Output','Turning Off All Motor Output',6('')];
END_VAR
(**)
(*Local Alarm*)
VAR
	tyAlmData : tyAlmDat;
	tyAlmData1 : tyAlmDat;
	tyAlmData2 : tyAlmDat;
	a_tyAlmText : ARRAY[10000..10199] OF tyAlmTxt := [(sAlmText:='Device Lost Connection',sRcyText:='Reset And Resume Operation.'),(sAlmText:='Device Removed Without Safety Remove. Please Restart PLC.',sRcyText:='Power Cycle Is Needed For USB Connectivity.'),(sAlmText:='Device Not Found.',sRcyText:='USB Without Safety Removed. Power Cycle Is Needed For USB Connectivity.'),(sAlmText:='Device Not Open.',sRcyText:='Frame Close Failed. Reset And Resume Operation.'),(sAlmText:='Device Not Connected. VID and PID Is Invalid',sRcyText:='Please Check The Vendor ID & Product ID.'),6((0)),(sAlmText:='Create User Directory Error',sRcyText:='An Error Occurred While Attempting To Create User Directory.Please Contact Nutek For A Possible Solution.'),(sAlmText:='Create Serial Directory Error',sRcyText:='An Error Occurred While Attempting To Create Serial Directory.Please Contact Nutek For A Possible Solution.'),(sAlmText:='Create USB Directory Error',sRcyText:='An Error Occurred While Attempting To Create USB Directory.Please Contact Nutek For A Possible Solution.'),(sAlmText:='Get Directory Info Error While Deleting Old Log',sRcyText:='An Error Was Encountered While Getting Directory Info. Please Contact Nutek For A Possible Solution.'),(sAlmText:='Directory Read Error While Deleting Old Log',sRcyText:='An Error Was Encountered While Reading Directory. Please Contact Nutek For A Possible Solution.'),(sAlmText:='File Delete Error While Deleting Old Log',sRcyText:='An Error Was Encountered While Trying To Delete File. Please Contact Nutek For A Possible Solution.'),(sAlmText:='File Open Error While Writing Serial Log',sRcyText:='An Error Was Encountered While Trying To Open File. Please Contact Nutek For A Possible Solution.'),(sAlmText:='File Create Error While Writing Serial Log',sRcyText:='An Error Was Encountered While Trying To Create File. Please Contact Nutek For A Possible Solution.'),(sAlmText:='Get File Info Error While Writing Serial Log',sRcyText:='An Error Was Encountered While Getting File Info. Please Contact Nutek For A Possible Solution.'),(sAlmText:='File Write Error While Writing Serial Log',sRcyText:='An Error Was Encountered While Trying To Write File. Please Contact Nutek For A Possible Solution.'),(sAlmText:='File Close Error While Writing Serial Log',sRcyText:='An Error Was Encountered While Trying To Close File. Please Contact Nutek For A Possible Solution.'),(sAlmText:='Directory Does Not Exist While Writing Serial Log',sRcyText:='The Directory Does Not Exist. Please Contact Nutek For A Possible Solution.'),177((0))];
END_VAR
(**)
(*Local Output*)
VAR
	sBarcodeOut : STRING[255];
END_VAR
(**)
(*Local Input*)
VAR
	udiRstErr : UDINT := 0;
	bPrep : BOOL := TRUE;
	bEn : BOOL := FALSE;
	bDis : BOOL := FALSE;
	bManual : BOOL := FALSE;
	sProgNm : STRING[15] := 'USBRdr';
	bNtSettingsLoadDone : BOOL := TRUE;
	uiVendorID : DINT := 16#05F9; (*1529*)
	uiProductID : DINT := 16#220C; (*8716*)
	bUSBRun : BOOL := FALSE;
	bScannerEn : BOOL := FALSE;
	dtCurrDT : DATE_AND_TIME := DT#1970-01-01-00:00:00;
	udiFileKeepDay : UDINT := 30;
END_VAR
(**)
(*Local*)
VAR
	bRstErr : BOOL;
	udiRstErrOld : UDINT;
	bInitDone : BOOL;
	bInitialDone : BOOL;
	fbGetUSBDevice : fbGetUSBDev;
	fbReadUSBDevice : fbReadUSBDev;
	fbRmvUSBDevice : fbSafetyRmvUSB;
	fbUSBTimer : TON := (PT:=T#5s);
	bUSBRmv : BOOL;
	bUSBDisconnected : BOOL;
	bNodeExist : BOOL;
END_VAR
(*Local Log file param*)
VAR
	usiStep : USINT;
	sDT : STRING[80];
	udiLogCntr : UDINT;
	udiWriteLogCntr : UDINT;
	iWriteLogStep : INT;
	dtCurrDTTemp : DATE_AND_TIME;
	a_sLogList : ARRAY[0..9] OF STRING[200];
	fbFileAppend1 : fbFileFullAppend;
	fbDirCreate1 : fbDirCreate;
	fbDirCreate2 : fbDirCreate;
	fbDirCreate3 : fbDirCreate;
	fbFileOldDel1 : fbFileOldDel;
	udiModuleNum : UDINT := 4601;
END_VAR
```

### Frame.var - Change By Project
```iecst
(*2019-05-29*)
(**)
(*Constant*)
VAR CONSTANT
	c_udiFrmHistoryMax : UDINT := 9;
END_VAR
(**)
(*Action & State & Status*)
VAR
	p_FrmStat : UDINT;
	p_FrmStatus : UDINT;
	p_FrmStatTxt : UDINT;
END_VAR
(**)
(*Alarm*)
VAR
	p_FrmAlmData : UDINT;
	p_FrmAlmData1 : UDINT;
END_VAR
(**)
(*Output*)
VAR
	p_FrmFullMsgRd : UDINT;
	p_FrmMsgRd : UDINT;
	p_FrmMsgRdValid : UDINT;
	p_FrmMsgRdLen : UDINT;
END_VAR
```

### Frame.typ - Change By Project
```iecst
(*2019-05-21*)
(**)
(*Action*)

TYPE
	eFrmAction :
		(
		FrmActIdle,
		FrmActFullWrite,
		FrmActFullRead,
		FrmActFullReadUntilValid,
		FrmActCreateDir,
		FrmActDeleteOldLog,
		FrmActAppendLog,
		FrmActBGStartLog,
		FrmActBGStopLog
		);
END_TYPE

(**)
(*Data*)
```

### Program Logical/RS232/DVFrame/Frame (IEC, version 1.00.0) - 1.00.0 - NtRecipe v5.00.0 , NtFileIO v5.00.0

#### Init.st - Change By Project
```iecst
(** 2019-05-29 **)
PROGRAM _INIT

	(* Always Change If Project Change *)

	//Pass Address To Global Address For External Use
	//Action, State & Status
	p_FrmStat		:= ADR(eStat);
	p_FrmStatus		:= ADR(eMainStatus);
	p_FrmStatTxt	:= ADR(sStatTxt);

	//Alarm
	p_FrmAlmData	:= ADR(tyAlmData);
	p_FrmAlmData1	:= ADR(tyAlmData1);
	//Output
	p_FrmFullMsgRd	:= ADR(sFullMsgRd);
	p_FrmMsgRd		:= ADR(sMsgRd);
	p_FrmMsgRdValid	:= ADR(bMsgRdValid);
	p_FrmMsgRdLen	:= ADR(uiMsgRdLen);

	(* Always Change If Project Change *)

END_PROGRAM
```

#### Act_InitGlobal.st - Change By Project
```iecst
(** 2019-05-10 **)
ACTION Act_InitGlobal:

	(* Always Change If Project Change *)

	//Pass Data To Link
	p_bLinkStartupRun ACCESS p_StartupRun;
	p_bLinkOpsRun ACCESS p_OpsRun;

	//Pass Data To Internal Use
	p_udiRstErr ACCESS p_RstErrReset;
	p_bPrep ACCESS p_NtParamRS232Prep;
	p_diStartCode1 ACCESS p_McParamRS232StartCode1;
	p_diStartCode2 ACCESS p_McParamRS232StartCode2;
	p_diEndCode1 ACCESS p_McParamRS232EndCode1;
	p_diEndCode2 ACCESS p_McParamRS232EndCode2;
	p_sProgNm ACCESS p_NtParamRS232ProgNm;
	p_bNtSettingsLoadDone ACCESS p_StartupNtSettingsLoadDone;
	p_dtCurrDT ACCESS p_TimeCurrDT;
	p_udiFileKeepDay ACCESS p_NtParamAlmFileKeepDay;

	(* Always Change If Project Change *)

END_ACTION
```

#### InputRef_Link.var - Change By Project
```iecst
(*2019-05-29*)
VAR
	p_bLinkStartupRun : REFERENCE TO BOOL;
END_VAR
(**)
VAR
	p_bLinkOpsRun : REFERENCE TO BOOL;
END_VAR
```

#### Act_LinkAction.st - Change By Project
```iecst
(** 2019-05-10 **)
ACTION Act_LinkAction:

	IF p_bLinkStartupRun = TRUE THEN
		p_eAct ACCESS p_StartupFrmAct;
	ELSE
		p_eAct ACCESS p_UIFrmAct; //Recipe Change by Barcode;

	END_IF

END_ACTION
```

#### Act_Link.st - Change By Project
```iecst
(** 2020-12-31 **)
ACTION Act_Link:

	//Default
	p_tyXOpenConfig.idle	:= 10;
	p_tyXOpenConfig.tx_cnt	:= 2;
	p_tyXOpenConfig.rx_cnt	:= 2;
	p_tyXOpenConfig.tx_len	:= 256;
	p_tyXOpenConfig.rx_len	:= 256;

	//End Code
	IF p_diEndCode1 <> -1 AND p_diEndCode2 <> -1 THEN

		p_tyXOpenConfig.delimc		:= 2;
		p_tyXOpenConfig.delim[0]	:= DINT_TO_USINT(p_diEndCode1);
		p_tyXOpenConfig.delim[1]	:= DINT_TO_USINT(p_diEndCode2);

	ELSIF p_diEndCode1 <> -1 AND p_diEndCode2 = -1 THEN

		p_tyXOpenConfig.delimc		:= 1;
		p_tyXOpenConfig.delim[0]	:= DINT_TO_USINT(p_diEndCode1);

	ELSIF p_diEndCode1 = -1 AND p_diEndCode2 <> -1 THEN

		p_tyXOpenConfig.delimc		:= 1;
		p_tyXOpenConfig.delim[0]	:= DINT_TO_USINT(p_diEndCode2);

	ELSIF p_diEndCode1 = -1 AND p_diEndCode2 = -1 THEN

		p_tyXOpenConfig.delimc		:= 0;

	END_IF

END_ACTION
```

#### Cyclic.st - Do Not Change!!!
```iecst
(** 2020-12-31 **)
PROGRAM _CYCLIC

	IF bInitDone = FALSE THEN
		bInitDone	:= TRUE;

		Act_InitLocal;
		Act_InitGlobal;

	ELSIF bInitialDone = FALSE THEN
		IF p_bNtSettingsLoadDone = TRUE THEN
			bInitialDone	:= TRUE;

			Act_Initial;
		END_IF

	ELSE

		Act_RstErr;
		Act_LinkAction;
		Act_Action;
		Act_LinkEn;

		IF (p_bPrep = TRUE) AND (p_bEn = TRUE) AND (p_bDis = FALSE) THEN
			Act_Link;
			Act_Background;
			Act_Main;
		ELSE
			IF eStat <> FrmActIdle THEN
				eStatus	:= Done;
			ELSE
				eStatus	:= Idle;
			END_IF
		END_IF

		Act_CombineErr;
		Act_Alarm;
		Act_Alarm1;

	END_IF

END_PROGRAM
```

#### Act_InitLocal.st - Do Not Change!!!
```iecst
(** 2019-05-20 **)
ACTION Act_InitLocal:

	//Input Reference Link To Local Variable
	p_eAct ACCESS ADR(eAct);
	p_udiRstErr ACCESS ADR(udiRstErr);
	p_bPrep ACCESS ADR(bPrep);
	p_bEn ACCESS ADR(bEn);
	p_bDis ACCESS ADR(bDis);

	p_sMsgWr ACCESS ADR(sMsgWr);
	p_tyParam ACCESS ADR(tyParam);
	p_tyXOpenConfig ACCESS ADR(tyXOpenConfig);
	p_diStartCode1 ACCESS ADR(diStartCode1);
	p_diStartCode2 ACCESS ADR(diStartCode2);
	p_diEndCode1 ACCESS ADR(diEndCode1);
	p_diEndCode2 ACCESS ADR(diEndCode2);
	p_sProgNm ACCESS ADR(sProgNm);
	p_dtCurrDT ACCESS ADR(dtCurrDT);
	p_udiFileKeepDay ACCESS ADR(udiFileKeepDay);
	p_bNtSettingsLoadDone ACCESS ADR(bNtSettingsLoadDone);

END_ACTION
```

#### Act_Initial.st - Do Not Change!!!
```iecst
(** 2019-05-21 **)
ACTION Act_Initial:

	//Initial
	sStatTxt	:= a_sStatText[eStat];

	fbFullWrite.tyCommParam		:= p_tyParam;
	fbFullWrite(bEn := FALSE);

	fbFullRead.tyCommParam		:= p_tyParam;
	fbFullRead.p_Data			:= ADR(sFullMsgRd);
	fbFullRead.uiMaxLen			:= SIZEOF(sFullMsgRd);
	fbFullRead(bEn := FALSE);

	fbFullReadUntilValid.tyCommParam	:= p_tyParam;
	fbFullReadUntilValid.p_Data			:= ADR(sFullMsgRd);
	fbFullReadUntilValid.uiMaxLen		:= SIZEOF(sFullMsgRd);
	fbFullReadUntilValid(bEn := FALSE);

	fbDirCreate1.sDevice	:= 'F';
	fbDirCreate1.sDirName	:= 'User';
	fbDirCreate1(bEn := FALSE);

	fbDirCreate2.sDevice	:= 'User';
	fbDirCreate2.sDirName	:= 'Serial';
	fbDirCreate2(bEn := FALSE);

	fbDirCreate3.sDevice	:= 'Serial';
	fbDirCreate3.sDirName	:= 'RS232';
	fbDirCreate3(bEn := FALSE);

	fbFileAppend1.sDevice	:= 'RS232';
	fbFileAppend1(bEn := FALSE);

	fbFileOldDel1.sDevice	:= 'RS232';
	fbFileOldDel1.sPath		:= '';
	fbFileOldDel1.sKeyword	:= 'Serial_';
	fbFileOldDel1(bEn := FALSE);

	fbFileRead1(bEn := FALSE);

END_ACTION
```

#### Act_Action.st - Do Not Change!!!
```iecst
(** 2019-05-22 **)
ACTION Act_Action:

	//Reset Error
	IF (eStatus = Error) AND bRstErr THEN
		p_eAct	:= FrmActIdle;
		eStat	:= FrmActIdle;
	END_IF

	//Set p_eAct
	IF eStatus = Idle OR eStatus = Busy OR eStatus = Done THEN
		eStat	:= p_eAct;
	END_IF

END_ACTION
```

#### Act_Main.st - Do Not Change!!!
```iecst
(** 2020-12-31 **)
ACTION Act_Main:

	//Main
	CASE eStat OF

		FrmActIdle:
			IF eStatus <> Idle THEN	//Reset Data
				//Private
				fbFullWrite(bEn := FALSE);
				fbFullRead(bEn := FALSE);
				fbFullReadUntilValid(bEn := FALSE);
				usiStep	:= 0;

				sStatTxt	:= a_sStatText[eStat];

			END_IF

			bMsgRdValid	:= FALSE;
			eStatus	:= Idle;

		FrmActFullRead:
			IF eStatus = Idle OR eStatus = Busy THEN

				eStatus	:= Busy;

				sStatTxt	:= a_sStatText[eStat];

				fbFullRead.tyXOpenConfig	:= p_tyXOpenConfig;
				fbFullRead(bEn := TRUE);
				IF fbFullRead.udiStatus = 0 THEN
					eStatus	:= Done;

					bMsgRdValid	:= fbFullRead.bReadValid;
					uiMsgRdLen	:= fbFullRead.uiLen;

					IF bMsgRdValid = TRUE THEN

						//Start Code
						IF p_diStartCode1 <> -1 AND p_diStartCode2 <> -1 THEN

							iStartCodeLen	:= 2;
							siStartCode1	:= DINT_TO_SINT(p_diStartCode1);
							siStartCode2	:= DINT_TO_SINT(p_diStartCode2);
							memmove(ADR(sStartCode) , ADR(siStartCode1) , 1);
							memmove(ADR(sStartCode) + 1 , ADR(siStartCode2) , 1);

							iStartCodePos	:= FIND(sFullMsgRd , sStartCode);

						ELSIF p_diStartCode1 <> -1 AND p_diStartCode2 = -1 THEN

							iStartCodeLen	:= 1;
							siStartCode1	:= DINT_TO_SINT(p_diStartCode1);
							memmove(ADR(sStartCode) , ADR(siStartCode1) , 1);

							iStartCodePos	:= FIND(sFullMsgRd , sStartCode);

						ELSIF p_diStartCode1 = -1 AND p_diStartCode2 <> -1 THEN

							iStartCodeLen	:= 1;
							siStartCode2	:= DINT_TO_SINT(p_diStartCode2);
							memmove(ADR(sStartCode) , ADR(siStartCode2) , 1);

							iStartCodePos	:= FIND(sFullMsgRd , sStartCode);

						ELSIF p_diStartCode1 = -1 AND p_diStartCode2 = -1 THEN

							iStartCodeLen	:= 0;
							iStartCodePos	:= 0;

						END_IF

						IF iStartCodePos <> 0 THEN
							sMsgRd	:= RIGHT(sFullMsgRd , (LEN(sFullMsgRd) - (iStartCodePos + iStartCodeLen - 1)));
						ELSIF iStartCodePos = 0 THEN
							sMsgRd	:= sFullMsgRd;	 //sMsgRd	:= ''; //Anson
						END_IF

						IF p_diEndCode1 <> -1 OR p_diEndCode2 <> -1 THEN
							sMsgRd	:= LEFT(sMsgRd , LEN(sMsgRd) - 1);
						END_IF

						fLogDTConvert(ADR(sDT) , p_dtCurrDT);
						memset(ADR(a_sLogList[udiLogCntr]) , 0 , SIZEOF(a_sLogList[udiLogCntr]));
						memcpy(ADR(a_sLogList[udiLogCntr]) + LEN(a_sLogList[udiLogCntr]) , ADR(sDT) , LEN(sDT));
						memcpy(ADR(a_sLogList[udiLogCntr]) + LEN(a_sLogList[udiLogCntr]) , ADR('$r$n') , LEN('$r$n'));
						memcpy(ADR(a_sLogList[udiLogCntr]) + LEN(a_sLogList[udiLogCntr]) , ADR('Received :') , LEN('Received :'));
						memcpy(ADR(a_sLogList[udiLogCntr]) + LEN(a_sLogList[udiLogCntr]) , ADR(sMsgRd) , LEN(sMsgRd));
						memcpy(ADR(a_sLogList[udiLogCntr]) + LEN(a_sLogList[udiLogCntr]) , ADR('$r$n$r$n') , LEN('$r$n$r$n'));

						udiLogCntr	:= udiLogCntr + 1;
						IF udiLogCntr = 10 THEN
							udiLogCntr	:= 0;
						END_IF

					END_IF

				ELSIF fbFullRead.udiStatus < 65534 THEN
					eStatus		:= Error;

					IF fbFullRead.udiStatus = 2350 THEN
						udiStatus	:= 10000;	//Open Port Error While Reading Message
					ELSIF fbFullRead.udiStatus = 2354 THEN
						udiStatus	:= 10001;	//Read Buffer Error While Reading Message
					ELSIF fbFullRead.udiStatus = 2355 THEN
						udiStatus	:= 10002;	//Release Receive Buffer Error While Reading Message
					ELSIF fbFullRead.udiStatus = 2356 THEN
						udiStatus	:= 10003;	//Close Port Error While Reading Message
					ELSE
						udiStatus	:= fbFullRead.udiStatus;
					END_IF

				END_IF

			END_IF

		FrmActFullWrite:
			IF eStatus = Idle OR eStatus = Busy THEN

				eStatus	:= Busy;

				sStatTxt	:= a_sStatText[eStat];

				fbFullWrite.tyXOpenConfig	:= p_tyXOpenConfig;
				fbFullWrite.p_Data			:= ADR(p_sMsgWr);
				fbFullWrite.uiLen			:= LEN(p_sMsgWr);
				fbFullWrite(bEn := TRUE);

				IF fbFullWrite.udiStatus = 0 THEN
					eStatus	:= Done;

					fLogDTConvert(ADR(sDT) , p_dtCurrDT);
					memset(ADR(a_sLogList[udiLogCntr]) , 0 , SIZEOF(a_sLogList[udiLogCntr]));
					memcpy(ADR(a_sLogList[udiLogCntr]) + LEN(a_sLogList[udiLogCntr]) , ADR(sDT) , LEN(sDT));
					memcpy(ADR(a_sLogList[udiLogCntr]) + LEN(a_sLogList[udiLogCntr]) , ADR('$r$n') , LEN('$r$n'));
					memcpy(ADR(a_sLogList[udiLogCntr]) + LEN(a_sLogList[udiLogCntr]) , ADR('Sent :') , LEN('Sent :'));
					memcpy(ADR(a_sLogList[udiLogCntr]) + LEN(a_sLogList[udiLogCntr]) , ADR(p_sMsgWr) , LEN(p_sMsgWr));
					memcpy(ADR(a_sLogList[udiLogCntr]) + LEN(a_sLogList[udiLogCntr]) , ADR('$r$n$r$n') , LEN('$r$n$r$n'));

					udiLogCntr	:= udiLogCntr + 1;
					IF udiLogCntr = 10 THEN
						udiLogCntr	:= 0;
					END_IF

				ELSIF fbFullWrite.udiStatus < 65534 THEN
					eStatus		:= Error;

					IF fbFullWrite.udiStatus = 2350 THEN
						udiStatus	:= 10004;	//Open Port Error While Writing Message
					ELSIF fbFullWrite.udiStatus = 2352 THEN
						udiStatus	:= 10005;	//Write Buffer Error While Writing Message
					ELSIF fbFullWrite.udiStatus = 2356 THEN
						udiStatus	:= 10006;	//Close Port Error While Writing Message
					ELSE
						udiStatus	:= fbFullWrite.udiStatus;
					END_IF
				END_IF

			END_IF

		FrmActFullReadUntilValid:
			IF eStatus = Idle OR eStatus = Busy THEN

				eStatus	:= Busy;

				sStatTxt	:= a_sStatText[eStat];

				fbFullReadUntilValid.tyXOpenConfig	:= p_tyXOpenConfig;
				fbFullReadUntilValid(bEn := TRUE);
				IF fbFullReadUntilValid.udiStatus = 0 THEN
					eStatus	:= Done;

					bMsgRdValid	:= TRUE;
					uiMsgRdLen	:= fbFullReadUntilValid.uiLen;

					IF bMsgRdValid = TRUE THEN

						//Start Code
						IF p_diStartCode1 <> -1 AND p_diStartCode2 <> -1 THEN

							iStartCodeLen	:= 2;
							siStartCode1	:= DINT_TO_SINT(p_diStartCode1);
							siStartCode2	:= DINT_TO_SINT(p_diStartCode2);
							memmove(ADR(sStartCode) , ADR(siStartCode1) , 1);
							memmove(ADR(sStartCode) + 1 , ADR(siStartCode2) , 1);

							iStartCodePos	:= FIND(sFullMsgRd , sStartCode);

						ELSIF p_diStartCode1 <> -1 AND p_diStartCode2 = -1 THEN

							iStartCodeLen	:= 1;
							siStartCode1	:= DINT_TO_SINT(p_diStartCode1);
							memmove(ADR(sStartCode) , ADR(siStartCode1) , 1);

							iStartCodePos	:= FIND(sFullMsgRd , sStartCode);

						ELSIF p_diStartCode1 = -1 AND p_diStartCode2 <> -1 THEN

							iStartCodeLen	:= 1;
							siStartCode2	:= DINT_TO_SINT(p_diStartCode2);
							memmove(ADR(sStartCode) , ADR(siStartCode2) , 1);

							iStartCodePos	:= FIND(sFullMsgRd , sStartCode);

						ELSIF p_diStartCode1 = -1 AND p_diStartCode2 = -1 THEN

							iStartCodeLen	:= 0;
							iStartCodePos	:= 0;

						END_IF

						IF iStartCodePos <> 0 THEN
							sMsgRd	:= RIGHT(sFullMsgRd , (LEN(sFullMsgRd) - (iStartCodePos + iStartCodeLen - 1)));
						ELSIF iStartCodePos = 0 THEN
							sMsgRd	:= sFullMsgRd;	 //sMsgRd	:= ''; //Anson
						END_IF

						IF p_diEndCode1 <> -1 OR p_diEndCode2 <> -1 THEN
							sMsgRd	:= LEFT(sMsgRd , LEN(sMsgRd) - 1);
						END_IF

						fLogDTConvert(ADR(sDT) , p_dtCurrDT);
						memset(ADR(a_sLogList[udiLogCntr]) , 0 , SIZEOF(a_sLogList[udiLogCntr]));
						memcpy(ADR(a_sLogList[udiLogCntr]) + LEN(a_sLogList[udiLogCntr]) , ADR(sDT) , LEN(sDT));
						memcpy(ADR(a_sLogList[udiLogCntr]) + LEN(a_sLogList[udiLogCntr]) , ADR('$r$n') , LEN('$r$n'));
						memcpy(ADR(a_sLogList[udiLogCntr]) + LEN(a_sLogList[udiLogCntr]) , ADR('Received :') , LEN('Received :'));
						memcpy(ADR(a_sLogList[udiLogCntr]) + LEN(a_sLogList[udiLogCntr]) , ADR(sMsgRd) , LEN(sMsgRd));
						memcpy(ADR(a_sLogList[udiLogCntr]) + LEN(a_sLogList[udiLogCntr]) , ADR('$r$n$r$n') , LEN('$r$n$r$n'));

						udiLogCntr	:= udiLogCntr + 1;
						IF udiLogCntr = 10 THEN
							udiLogCntr	:= 0;
						END_IF
					END_IF

				ELSIF fbFullReadUntilValid.udiStatus < 65534 THEN
					eStatus		:= Error;
					bMsgRdValid	:= FALSE;

					IF fbFullReadUntilValid.udiStatus = 2350 THEN
						udiStatus	:= 10007;	//Open Port Error While Reading Message
					ELSIF fbFullReadUntilValid.udiStatus = 2354 THEN
						udiStatus	:= 10008;	//Read Buffer Error While Reading Message
					ELSIF fbFullReadUntilValid.udiStatus = 2355 THEN
						udiStatus	:= 10009;	//Release Receive Buffer Error While Reading Message
					ELSIF fbFullReadUntilValid.udiStatus = 2356 THEN
						udiStatus	:= 10010;	//Close Port Error While Reading Message
					ELSE
						udiStatus	:= fbFullReadUntilValid.udiStatus;
					END_IF

				END_IF

			END_IF

		FrmActCreateDir:
			IF eStatus = Idle OR eStatus = Busy THEN

				eStatus	:= Busy;

				sStatTxt	:= a_sStatText[eStat];

				CASE usiStep OF
					0:
						fbDirCreate1(bEn := TRUE);
						IF fbDirCreate1.udiStatus = 0 THEN
							usiStep	:= 1;
						ELSIF fbDirCreate1.udiStatus < 65534 THEN
							eStatus		:= Error;

							IF fbDirCreate1.udiStatus = 1908 THEN
								udiStatus	:= 10011;	//Create User Directory Error
							ELSE
								udiStatus	:= fbDirCreate1.udiStatus;
							END_IF
						END_IF

					1:
						fbDirCreate2(bEn := TRUE);
						IF fbDirCreate2.udiStatus = 0 THEN
							usiStep	:= 2;
						ELSIF fbDirCreate2.udiStatus < 65534 THEN
							eStatus		:= Error;

							IF fbDirCreate2.udiStatus = 1908 THEN
								udiStatus	:= 10012;	//'Create Serial Directory Error'
							ELSE
								udiStatus	:= fbDirCreate2.udiStatus;
							END_IF
						END_IF
					2:
						fbDirCreate3(bEn := TRUE);
						IF fbDirCreate3.udiStatus = 0 THEN
							eStatus	:= Done;
						ELSIF fbDirCreate3.udiStatus < 65534 THEN
							eStatus		:= Error;

							IF fbDirCreate3.udiStatus = 1908 THEN
								udiStatus	:= 10013;	//'Create RS232 Directory Error'
							ELSE
								udiStatus	:= fbDirCreate3.udiStatus;
							END_IF
						END_IF
				END_CASE

			END_IF

		FrmActDeleteOldLog:
			IF eStatus = Idle OR eStatus = Busy THEN

				eStatus	:= Busy;

				sStatTxt	:= a_sStatText[eStat];

				fbFileOldDel1.dtDTNow			:= p_dtCurrDT;
				fbFileOldDel1.udiFileKeepDay	:= p_udiFileKeepDay;
				fbFileOldDel1(bEn := TRUE);
				IF fbFileOldDel1.udiStatus = 0 THEN
					eStatus	:= Done;
				ELSIF fbFileOldDel1.udiStatus < 65534 THEN
					eStatus		:= Error;

					IF fbFileOldDel1.udiStatus = 1910 THEN
						udiStatus	:= 10014;	//Get Directory Info Error While Deleting Old Log
					ELSIF fbFileOldDel1.udiStatus = 1911 THEN
						udiStatus	:= 10015;	//Directory Read Error While Deleting Old Log
					ELSIF fbFileOldDel1.udiStatus = 1912 THEN
						udiStatus	:= 10016;	//File Delete Error While Deleting Old Log
					ELSE
						udiStatus	:= fbFileOldDel1.udiStatus;
					END_IF
				END_IF

			END_IF

		FrmActAppendLog:
			IF eStatus = Idle OR eStatus = Busy THEN

				eStatus	:= Busy;

				sStatTxt	:= a_sStatText[eStat];

				dtCurrDTTemp			:= p_dtCurrDT;
				fbFileAppend1.sFile		:= DT_TO_STRING(dtCurrDTTemp);
				fbFileAppend1.sFile		:= MID(fbFileAppend1.sFile , 10 , 4);
				fbFileAppend1.sFile		:= CONCAT('Serial_' , fbFileAppend1.sFile);
				fbFileAppend1.sFile		:= CONCAT(fbFileAppend1.sFile , '.dat');

				fbFileAppend1.p_Src		:= ADR(a_sLogList[udiWriteLogCntr]);
				fbFileAppend1.udiLen	:= LEN(a_sLogList[udiWriteLogCntr]);

				fbFileAppend1(bEn := TRUE);
				IF fbFileAppend1.udiStatus = 0 THEN
					IF udiWriteLogCntr >= udiLogCntr THEN
						eStatus	:= Done;
					ELSE
						udiWriteLogCntr	:= udiWriteLogCntr + 1;
						fbFileAppend1(bEn := FALSE);
					END_IF

				ELSIF fbFileAppend1.udiStatus < 65534 THEN
					eStatus		:= Error;

					IF fbFileAppend1.udiStatus = 1900 THEN
						udiStatus	:= 10017;	//File Open Error While Writing Serial Log
					ELSIF fbFileAppend1.udiStatus = 1901 THEN
						udiStatus	:= 10018;	//File Create Error While Writing Serial Log
					ELSIF fbFileAppend1.udiStatus = 1913 THEN
						udiStatus	:= 10019;	//Get File Info Error While Writing Serial Log
					ELSIF fbFileAppend1.udiStatus = 1903 THEN
						udiStatus	:= 10020;	//File Write Error While Writing Serial Log
					ELSIF fbFileAppend1.udiStatus = 1904 THEN
						udiStatus	:= 10021;	//File Close Error While Writing Serial Log
					ELSIF fbFileAppend1.udiStatus = 1914 THEN
						udiStatus	:= 10022;	//Directory Does Not Exist While Writing Serial Log
					ELSE
						udiStatus	:= fbFileAppend1.udiStatus;
					END_IF
				END_IF

			END_IF

		FrmActBGStartLog:
			IF eStatus = Idle OR eStatus = Busy THEN

				sStatTxt	:= a_sStatText[eStat];

				bFrmLog		:= TRUE;
				eStatus		:= Done;

			END_IF

		FrmActBGStopLog:
			IF eStatus = Idle OR eStatus = Busy THEN

				sStatTxt	:= a_sStatText[eStat];

				bFrmLog		:= FALSE;
				eStatus		:= Done;

			END_IF

	END_CASE

END_ACTION
```

#### Act_Background.st - Do Not Change!!!
```iecst
(** 2019-05-21 **)
ACTION Act_Background:

	//End Code
	IF p_diEndCode1 <> -1 AND p_diEndCode2 <> -1 THEN

		p_tyXOpenConfig.delimc		:= 2;
		p_tyXOpenConfig.delim[0]	:= DINT_TO_USINT(p_diEndCode1);
		p_tyXOpenConfig.delim[1]	:= DINT_TO_USINT(p_diEndCode2);

	ELSIF p_diEndCode1 <> -1 AND p_diEndCode2 = -1 THEN

		p_tyXOpenConfig.delimc		:= 1;
		p_tyXOpenConfig.delim[0]	:= DINT_TO_USINT(p_diEndCode1);

	ELSIF p_diEndCode1 = -1 AND p_diEndCode2 <> -1 THEN

		p_tyXOpenConfig.delimc		:= 1;
		p_tyXOpenConfig.delim[0]	:= DINT_TO_USINT(p_diEndCode2);

	ELSIF p_diEndCode1 = -1 AND p_diEndCode2 = -1 THEN

		p_tyXOpenConfig.delimc		:= 0;

	END_IF

	IF (eStatus1 = Error) AND bRstErr THEN
		eStatus1	:= Idle;
		udiStatus1	:= 0;

		fbFileAppend1(bEn := FALSE);
		iWriteLogStep	:= 0;
	END_IF

	IF eStatus1 <> Error THEN

		IF udiWriteLogCntr <> udiLogCntr THEN

			CASE iWriteLogStep OF

				0:
					dtCurrDTTemp			:= p_dtCurrDT;
					fbFileAppend1.sFile		:= DT_TO_STRING(dtCurrDTTemp);
					fbFileAppend1.sFile		:= MID(fbFileAppend1.sFile , 10 , 4);
					fbFileAppend1.sFile		:= CONCAT('_' , fbFileAppend1.sFile);
					fbFileAppend1.sFile		:= CONCAT('Serial' , fbFileAppend1.sFile);
					fbFileAppend1.sFile		:= CONCAT(fbFileAppend1.sFile , '.dat');

					fbFileAppend1.p_Src		:= ADR(a_sLogList[udiWriteLogCntr]);
					fbFileAppend1.udiLen	:= LEN(a_sLogList[udiWriteLogCntr]);

					iWriteLogStep	:= 1;

				1:
					fbFileAppend1(bEn := TRUE);
					IF fbFileAppend1.udiStatus = 0 THEN
						fbFileAppend1(bEn := FALSE);

						udiWriteLogCntr	:= udiWriteLogCntr + 1;
						IF udiWriteLogCntr = 10 THEN
							udiWriteLogCntr	:= 0;
						END_IF

						iWriteLogStep	:= 0;

					ELSIF fbFileAppend1.udiStatus < 65534 THEN
						eStatus1	:= Error;

						IF fbFileAppend1.udiStatus = 1900 THEN
							udiStatus1	:= 10017;	//File Open Error While Writing Serial Log
						ELSIF fbFileAppend1.udiStatus = 1901 THEN
							udiStatus1	:= 10018;	//File Create Error While Writing Serial Log
						ELSIF fbFileAppend1.udiStatus = 1913 THEN
							udiStatus1	:= 10019;	//Get File Info Error While Writing Serial Log
						ELSIF fbFileAppend1.udiStatus = 1903 THEN
							udiStatus1	:= 10020;	//File Write Error While Writing Serial Log
						ELSIF fbFileAppend1.udiStatus = 1904 THEN
							udiStatus1	:= 10021;	//File Close Error While Writing Serial Log
						ELSIF fbFileAppend1.udiStatus = 1914 THEN
							udiStatus1	:= 10022;	//Directory Does Not Exist While Writing Serial Log
						ELSE
							udiStatus1	:= fbFileAppend1.udiStatus;
						END_IF

						iWriteLogStep	:= 0;

					END_IF

			END_CASE

		END_IF

	END_IF

	IF bShareFolderEn THEN
		DevLink_0.enable 	:= TRUE;
		DevLink_0.pDevice 	:= ADR(sFileLocation);
		DevLink_0.pParam	:= ADR('/SIP=192.168.0.220 /PROTOCOL=cifs /SHARE=ThisPath /USER=jiunloh /PASSWORD=Chaos@2013 /DOMAIN=NUTEKSG ');

		ErrorCode := FileIoGetSysError();

		DevLink_0();

		bFolderValid:= DevLink_0.status=20730;

		IF bFolderValid THEN
			bShareFolderEn := FALSE;
		END_IF
	END_IF

	IF bFolderValid THEN

		fbFileRead1.sDevice		:= sFileLocation;
		fbFileRead1.sFile		:= '888.txt';
		fbFileRead1.udiOffset	:= 0;
		fbFileRead1.p_Dest		:= ADR(sFileData);
		fbFileRead1.udiLen		:= SIZEOF(sFileData);
		fbFileRead1(bEn := TRUE);

		IF fbFileRead1.udiStatus = 0 THEN
			bFileDataRead := TRUE;
			bFolderValid := FALSE;
		END_IF

	END_IF

END_ACTION
```

#### Act_Alarm.st - Do Not Change!!!
```iecst
(** 2019-03-25 **)
ACTION Act_Alarm:

	//Error
	IF EDGEPOS(eStatus = Error) THEN

		tyAlmData.sProgNm		:= p_sProgNm;
		tyAlmData.udiCode		:= udiStatus;
		tyAlmData.eSeverity		:= AlmSeverityError;
		tyAlmData.udiRunTime	:= tyAlmData.udiRunTime + 1;
		tyAlmData.bAlm			:= TRUE;
		tyAlmData.udiModuleNum  := udiModuleNum;
		g_sFrameProgNm			:= p_sProgNm;

		//Get Error Message
		IF tyAlmData.udiCode < 10000 OR tyAlmData.udiCode > 10099 THEN
			tyAlmData.sAlmMsg	:= 'Unknown';
			tyAlmData.sRcyMsg	:= 'Unknown';
		ELSE
			tyAlmData.sAlmMsg	:= a_tyAlmText[tyAlmData.udiCode].sAlmText;
			tyAlmData.sRcyMsg	:= a_tyAlmText[tyAlmData.udiCode].sRcyText;
		END_IF

		sStatTxt	:= tyAlmData.sAlmMsg;

	ELSIF bRstErr AND (tyAlmData.udiCode <> 0) THEN

		tyAlmData.udiCode	:= 0;
		tyAlmData.eSeverity	:= AlmSeverityNA;
		tyAlmData.sAlmMsg	:= '';
		tyAlmData.sRcyMsg	:= '';
		tyAlmData.bAlm			:=  FALSE;
		sStatTxt	:= a_sStatText[eStat];

	END_IF

END_ACTION
```

#### Act_Alarm1.st - Do Not Change!!!
```iecst
(** 2019-03-25 **)
ACTION Act_Alarm1:

	//Error
	IF EDGEPOS(eStatus1 = Error) THEN

		tyAlmData1.sProgNm		:= p_sProgNm;
		tyAlmData1.udiCode		:= udiStatus1;
		tyAlmData1.eSeverity	:= AlmSeverityError;
		tyAlmData1.udiRunTime	:= tyAlmData1.udiRunTime + 1;
		tyAlmData1.bAlm			:= TRUE;
		tyAlmData1.udiModuleNum  := udiModuleNum;
		g_sFrameProgNm			:= p_sProgNm;

		//Get Error Message
		IF tyAlmData1.udiCode < 10000 OR tyAlmData1.udiCode > 10199 THEN
			tyAlmData1.sAlmMsg	:= 'Unknown';
			tyAlmData1.sRcyMsg	:= 'Unknown';
		ELSE
			tyAlmData1.sAlmMsg	:= a_tyAlmText[tyAlmData1.udiCode].sAlmText;
			tyAlmData1.sRcyMsg	:= a_tyAlmText[tyAlmData1.udiCode].sRcyText;
		END_IF

		sStatTxt	:= tyAlmData1.sAlmMsg;

	ELSIF bRstErr AND (tyAlmData1.udiCode <> 0) THEN

		tyAlmData1.udiCode		:= 0;
		tyAlmData1.eSeverity	:= AlmSeverityNA;
		tyAlmData1.sAlmMsg		:= '';
		tyAlmData1.sRcyMsg		:= '';
		tyAlmData1.bAlm			:= FALSE;
		sStatTxt	:= a_sStatText[eStat];

	END_IF

END_ACTION
```

#### InputRef.var - Do Not Change!!!
```iecst
(*2019-05-29*)
(**)
(*General*)
VAR
	p_eAct : REFERENCE TO eFrmAction;
	p_udiRstErr : REFERENCE TO UDINT;
	p_bPrep : REFERENCE TO BOOL;
	p_bEn : REFERENCE TO BOOL;
	p_bDis : REFERENCE TO BOOL;
END_VAR
(**)
(*Configuration*)
VAR
	p_sMsgWr : REFERENCE TO STRING[80];
	p_tyParam : REFERENCE TO tyFrmParam;
	p_tyXOpenConfig : REFERENCE TO XOPENCONFIG;
	p_diStartCode1 : REFERENCE TO DINT;
	p_diStartCode2 : REFERENCE TO DINT;
	p_diEndCode1 : REFERENCE TO DINT;
	p_diEndCode2 : REFERENCE TO DINT;
	p_sProgNm : REFERENCE TO STRING[15];
	p_bNtSettingsLoadDone : REFERENCE TO BOOL;
	p_dtCurrDT : REFERENCE TO DATE_AND_TIME;
	p_udiFileKeepDay : REFERENCE TO UDINT;
END_VAR
```

#### Local.var - Do Not Change!!!
```iecst
(*2019-05-29*)
(**)
(*Local Action, State & Status*)
VAR
	eAct : eFrmAction := FrmActIdle;
	eStat : eFrmAction := FrmActIdle;
	eMainStatus : eFBStatus := Idle;
	eStatus : eFBStatus := Idle;
	eStatus1 : eFBStatus := Idle;
	udiStatus : UDINT := 0;
	udiStatus1 : UDINT := 0;
	sStatTxt : STRING[200] := '';
	a_sStatText : ARRAY[0..50] OF STRING[200] := ['Idling','Writing RS232','Reading RS232','Reading RS232 Until Data Valid','Creating Directory','Deleting Old Alarm Log File','Appending Alarm Log File','Background Start Alarm Log','Background Stop Alarm Log',42('')];
END_VAR
(**)
(*Local Alarm*)
VAR
	tyAlmData : tyAlmDat;
	tyAlmData1 : tyAlmDat;
	a_tyAlmText : ARRAY[10000..10099] OF tyAlmTxt := [(sAlmText:='Open Port Error While Reading Message',sRcyText:='Check Hardware Condition. Contact Nutek For Possible Solution.'),(sAlmText:='Read Buffer Error While Reading Message',sRcyText:='Check Hardware Condition. Contact Nutek For Possible Solution.'),(sAlmText:='Release Receive Buffer Error While Reading Message',sRcyText:='Check Hardware Condition. Contact Nutek For Possible Solution.'),(sAlmText:='Close Port Error While Reading Message',sRcyText:='Check Hardware Condition. Contact Nutek For Possible Solution.'),(sAlmText:='Open Port Error While Writing Message',sRcyText:='Check Hardware Condition. Contact Nutek For Possible Solution.'),(sAlmText:='Write Buffer Error While Writing Message',sRcyText:='Check Hardware Condition. Contact Nutek For Possible Solution.'),(sAlmText:='Close Port Error While Writing Message',sRcyText:='Check Hardware Condition. Contact Nutek For Possible Solution.'),(sAlmText:='Open Port Error While Reading Message',sRcyText:='Check Hardware Condition. Contact Nutek For Possible Solution.'),(sAlmText:='Read Buffer Error While Reading Message',sRcyText:='Check Hardware Condition. Contact Nutek For Possible Solution.'),(sAlmText:='Release Receive Buffer Error While Reading Message',sRcyText:='Check Hardware Condition. Contact Nutek For Possible Solution.'),(sAlmText:='Close Port Error While Reading Message',sRcyText:='Check Hardware Condition. Contact Nutek For Possible Solution.'),(sAlmText:='Create User Directory Error',sRcyText:='An Error Occurred While Attempting To Create User Directory. Please Contact Nutek For A Possible Solution'),(sAlmText:='Create Serial Directory Error',sRcyText:='An Error Occurred While Attempting To Create Serial Directory. Please Contact Nutek For A Possible Solution'),(sAlmText:='Create RS232 Directory Error',sRcyText:='An Error Occurred While Attempting To Create RS232 Directory. Please Contact Nutek For A Possible Solution.'),(sAlmText:='Get Directory Info Error While Deleting Old Log',sRcyText:='An Error Was Encountered While Getting Directory Info. Please Contact Nutek For A Possible Solution.'),(sAlmText:='Directory Read Error While Deleting Old Log',sRcyText:='An Error Was Encountered While Reading Directory. Please Contact Nutek For A Possible Solution.'),(sAlmText:='File Delete Error While Deleting Old Log',sRcyText:='An Error Was Encountered While Trying To Delete File. Please Contact Nutek For A Possible Solution.'),(sAlmText:='File Open Error While Writing Serial Log',sRcyText:='An Error Was Encountered While Trying To Open File. Please Contact Nutek For A Possible Solution.'),(sAlmText:='File Create Error While Writing Serial Log',sRcyText:='An Error Was Encountered While Trying To Create File. Please Contact Nutek For A Possible Solution.'),(sAlmText:='Get File Info Error While Writing Serial Log',sRcyText:='An Error Was Encountered While Getting File Info. Please Contact Nutek For A Possible Solution.'),(sAlmText:='File Write Error While Writing Serial Log',sRcyText:='An Error Was Encountered While Trying To Write File. Please Contact Nutek For A Possible Solution.'),(sAlmText:='File Close Error While Writing Serial Log',sRcyText:='An Error Was Encountered While Trying To Close File. Please Contact Nutek For A Possible Solution.'),(sAlmText:='Directory Does Not Exist While Writing Serial Log',sRcyText:='The Directory Does Not Exist. Please Contact Nutek For A Possible Solution.'),77((0))];
END_VAR
(**)
(*Local Output*)
VAR
	sFullMsgRd : STRING[80];
	sMsgRd : STRING[80];
	bMsgRdValid : BOOL;
	uiMsgRdLen : UINT;
END_VAR
(**)
(*Local Input*)
VAR
	udiRstErr : UDINT := 0;
	bPrep : BOOL := TRUE;
	bEn : BOOL := TRUE;
	bDis : BOOL := FALSE;
	sMsgWr : STRING[80];
	tyParam : tyFrmParam;
	tyXOpenConfig : XOPENCONFIG := (idle:=10,tx_cnt:=2,rx_cnt:=2,tx_len:=256,rx_len:=256);
	diStartCode1 : DINT;
	diStartCode2 : DINT;
	diEndCode1 : DINT;
	diEndCode2 : DINT;
	dtCurrDT : DATE_AND_TIME;
	udiFileKeepDay : UDINT := 30;
	dtCurrDTTemp : DATE_AND_TIME;
	sProgNm : STRING[15] := 'RS232';
	bNtSettingsLoadDone : BOOL := TRUE;
END_VAR
(**)
(*Local*)
VAR
	ErrorCode : UINT;
	DevLink_0 : DevLink;
	bFileDataRead : BOOL;
	bBuildIn : BOOL;
	bFolderValid : BOOL;
	bShareFolderEn : BOOL;
	bRstErr : BOOL;
	udiRstErrOld : UDINT;
	bInitDone : BOOL;
	bInitialDone : BOOL;
	fbFullWrite : fbFrmFullWrite;
	fbFullRead : fbFrmFullRead;
	fbFullReadUntilValid : fbFrmFullReadUntilValid;
	iStartCodeLen : INT;
	siStartCode1 : SINT;
	siStartCode2 : SINT;
	sStartCode : STRING[2];
	iStartCodePos : INT;
	usiStep : USINT;
	sDT : STRING[80];
	bFrmLog : BOOL;
	iWriteLogStep : INT := 0;
	udiLogCntr : UDINT;
	udiWriteLogCntr : UDINT;
	a_sLogList : ARRAY[0..c_udiFrmHistoryMax] OF STRING[200];
	fbFileAppend1 : fbFileFullAppend;
	fbFileAppend2 : fbFileFullAppend;
	fbDirCreate1 : fbDirCreate;
	fbDirCreate2 : fbDirCreate;
	fbDirCreate3 : fbDirCreate;
	fbFileRead1 : fbFileFullRead;
	sFileLocation : STRING[254] := '123';
	sFileData : STRING[254];
	fbFileOldDel1 : fbFileOldDel;
	udiModuleNum : UDINT := 6211;
END_VAR
```

### Program Logical/MtrPshr/MtrPshr

#### InputRef.var
```iecst
(*2019-03-25*)
(**)
(*General*)
VAR
	p_eAct : REFERENCE TO eMtrPshrAction;
	p_udiRstErr : REFERENCE TO UDINT;
	p_bPrep : REFERENCE TO BOOL;
	p_bEn : REFERENCE TO BOOL;
	p_bDis : REFERENCE TO BOOL;
END_VAR
(**)
(*Configuration*)
VAR
	p_bManual : REFERENCE TO BOOL;
	p_bDir : REFERENCE TO BOOL;
	p_tAlmRstTm : REFERENCE TO TIME;
	p_tAlmTrigTm : REFERENCE TO TIME;
	p_tMtrBrkOffDlyTm : REFERENCE TO TIME;
	p_tExtTO : REFERENCE TO TIME;
	p_tRetTO : REFERENCE TO TIME;
	p_diExtSlowSpd : REFERENCE TO DINT;
	p_diRetSlowSpd : REFERENCE TO DINT;
	p_diExtNomSpd : REFERENCE TO DINT;
	p_diRetNomSpd : REFERENCE TO DINT;
	p_diExtTorque : REFERENCE TO DINT;
	p_diRetTorque : REFERENCE TO DINT;
	p_diStartTorque : REFERENCE TO DINT;
	p_sProgNm : REFERENCE TO STRING[15];
	p_bNtSettingsLoadDone : REFERENCE TO BOOL;
END_VAR
(**)
(*Input*)
VAR
	p_bExtSen : REFERENCE TO BOOL;
	p_bRetSen : REFERENCE TO BOOL;
	p_bExtSlowSen : REFERENCE TO BOOL;
	p_bRetSlowSen : REFERENCE TO BOOL;
	p_bExtSafetySen : REFERENCE TO BOOL;
	p_bRetSafetySen : REFERENCE TO BOOL;
	p_bAlarmSig : REFERENCE TO BOOL;
	p_bTorqueSig : REFERENCE TO BOOL;
END_VAR
```

#### InputRef_Link.var
```iecst
(*2019-04-09*)
(**)
VAR
	p_bLinkOpsRun : REFERENCE TO BOOL;
END_VAR
(**)
VAR
	p_bLinkDISafetyRlySig : REFERENCE TO BOOL;
	p_bLinkPullConvPullerExtCtrl : REFERENCE TO BOOL;
	p_bLinkPullConvPullerRetCtrl : REFERENCE TO BOOL;
	p_bLinkAlarmSig : REFERENCE TO BOOL;
END_VAR
```

#### Local.var
```iecst
(*2019-06-17*)
(**)
(*Local Action, State & Status*)
VAR
	eAct : eMtrPshrAction := MtrPshrActIdle;
	eStat : eMtrPshrAction := MtrPshrActIdle;
	eStatus : eFBStatus := Idle;
	udiStatus : UDINT := 0;
	sStatTxt : STRING[200] := '';
	a_sStatText : ARRAY[0..60] OF STRING[200] := ['Idling','Extending','Retracting','Stopping','Turning On Motor Extend','Turning Off Motor Extend','Turning On Motor Retract','Turning Off Motor Retract','Turning On Speed Binary Bit 0','Turning Off Speed Binary Bit 0','Turning On Speed Binary Bit 1','Turning Off Speed Binary Bit 1','Turning On Speed Binary Bit 2','Turning Off Speed Binary Bit 2','Turning On Signal On','Turning Off Signal On','Turning On Brake','Turning Off Brake','Turning On Alarm Reset','Turning Off Alarm Reset','Turning On All Motor Output','Turning Of All Motor Output',39('')];
END_VAR
(**)
(*Local Alarm*)
VAR
	tyAlmData : tyAlmDat;
	a_tyAlmText : ARRAY[10000..10199] OF tyAlmTxt := [(sAlmText:='Pusher Retract Sensor Off Time Out In Extend Check While Pusher Extend',sRcyText:='Sensor Timeout Expired Before Operation Completed. Sensor Operation Is Abnormal. Solve The Error To Resume Operation.'),(sAlmText:='Pusher Extend Sensor On Time Out In Extend Check While Pusher Extend',sRcyText:='Sensor Timeout Expired Before Operation Completed. Sensor Operation Is Abnormal. Solve The Error To Resume Operation.'),(sAlmText:='Pusher Extend Safety Sensor Error In Extend Check While Pusher Extend',sRcyText:='Safety System Has Been Triggered. All Operations Are Disable. Remove the Obstacle That Triggered The Safety Interlock To Resume Operation.'),(sAlmText:='Pusher Extend Sensor Off Time Out In Retract Check While Pusher Retract',sRcyText:='Sensor Timeout Expired Before Operation Completed. Sensor Operation Is Abnormal. Solve The Error To Resume Operation.'),(sAlmText:='Pusher Retract Sensor On Time Out In Retract Check While Pusher Retract',sRcyText:='Sensor Timeout Expired Before Operation Completed. Sensor Operation Is Abnormal. Solve The Error To Resume Operation.'),(sAlmText:='Pusher Retract Safety Sensor Error In Retract Check While Pusher Retract',sRcyText:='Safety System Has Been Triggered. All Operations Are Disable. Remove the Obstacle That Triggered The Safety Interlock To Resume Operation.'),(sAlmText:='Motorized Puller Alarm Occur',sRcyText:='Motorized Puller Operated Abnormal. Reset The Error To Resume Operation. If The Problem Persists, Please Contact Nutek For A Possible Solution.'),193((sAlmText:='',sRcyText:=''))];
END_VAR
(**)
(*Local Output*)
VAR
	bExtended : BOOL;
	bRetracted : BOOL;
	bCW : BOOL;
	bCCW : BOOL;
	bSpdBinBit0 : BOOL;
	bSpdBinBit1 : BOOL;
	bSpdBinBit2 : BOOL;
	bSigOn : BOOL;
	bBrake : BOOL;
	bAlmRst : BOOL;
END_VAR
(**)
(*Local Input*)
VAR
	udiRstErr : UDINT := 0;
	bPrep : BOOL := TRUE;
	bEn : BOOL := TRUE;
	bDis : BOOL := FALSE;
	bManual : BOOL := FALSE;
	bDir : BOOL := FALSE;
	tAlmRstTm : TIME := T#1s;
	tAlmTrigTm : TIME := T#1s;
	tMtrBrkOffDlyTm : TIME := T#500ms;
	tExtTO : TIME := T#20s;
	tRetTO : TIME := T#20s;
	diExtSlowSpd : DINT;
	diRetSlowSpd : DINT;
	diExtNomSpd : DINT;
	diRetNomSpd : DINT;
	diExtTorque : DINT;
	diRetTorque : DINT;
	diStartTorque : DINT;
	bExtSen : BOOL;
	bRetSen : BOOL;
	bExtSlowSen : BOOL;
	bRetSlowSen : BOOL;
	bExtSafetySen : BOOL := TRUE;
	bRetSafetySen : BOOL := TRUE;
	bAlarmSig : BOOL;
	bTorqueSig : BOOL;
	sProgNm : STRING[15] := 'MtrPshr';
	bNtSettingsLoadDone : BOOL := TRUE;
END_VAR
(**)
(*Local*)
VAR
	bRstErr : BOOL;
	udiRstErrOld : UDINT;
	bInitDone : BOOL;
	bInitialDone : BOOL;
	eStatOld : eMtrPshrAction := MtrPshrActIdle;
	iAnalogTorque : INT;
	diMtrSpd : DINT;
	bMtrSpdSlw : BOOL;
	fbAlmRstTm : TON := (PT:=T#1s);
	fbAlmTrigTm : TON := (PT:=T#2s);
	fbMtrBrkOffDlyTm : TON;
	fbMtrPshrExtChk : fbPneuExtRetSenExtChk;
	fbMtrPshrRetChk : fbPneuExtRetSenRetChk;
	usiPercent : USINT := 100;
	iMtrVolt : INT := 16800;
	iRetSlwTor : INT := 6300;
	udiModuleNum : UDINT := 6261;
END_VAR
```

#### Act_Alarm.st
```iecst
(** 2019-03-25 **)
ACTION Act_Alarm:

	//Error
	IF EDGEPOS(eStatus = Error) THEN

		tyAlmData.sProgNm		:= p_sProgNm;
		tyAlmData.udiCode		:= udiStatus;
		tyAlmData.eSeverity		:= AlmSeverityError;
		tyAlmData.udiRunTime	:= tyAlmData.udiRunTime + 1;
		tyAlmData.bAlm			:= TRUE;
		tyAlmData.udiModuleNum  := udiModuleNum;
		g_sMtrPshrProgNm		:= p_sProgNm;

		//Get Error Message
		IF tyAlmData.udiCode < 10000 OR tyAlmData.udiCode > 10199 THEN
			tyAlmData.sAlmMsg	:= 'Unknown';
			tyAlmData.sRcyMsg	:= 'Unknown';
		ELSE
			tyAlmData.sAlmMsg	:= a_tyAlmText[tyAlmData.udiCode].sAlmText;
			tyAlmData.sRcyMsg	:= a_tyAlmText[tyAlmData.udiCode].sRcyText;
		END_IF

		sStatTxt	:= tyAlmData.sAlmMsg;

	ELSIF bRstErr AND (tyAlmData.udiCode <> 0) THEN

		tyAlmData.udiCode	:= 0;
		tyAlmData.eSeverity	:= AlmSeverityNA;
		tyAlmData.sAlmMsg	:= '';
		tyAlmData.sRcyMsg	:= '';
		tyAlmData.bAlm			:= FALSE;
		sStatTxt	:= a_sStatText[eStat];

	END_IF

END_ACTION
```

#### Act_Background.st
```iecst
(** 2019-01-18 **)
ACTION Act_Background:

	IF p_bExtSen = FALSE THEN
		bExtended	:= FALSE;
	END_IF

	IF p_bRetSen = FALSE THEN
		bRetracted	:= FALSE;
	END_IF

	//Torque Minimum Value
	IF iAnalogTorque < 1500 THEN
		iAnalogTorque	:= 1500;
	END_IF

	//Abnormal Movement
	IF eStatus <> Error THEN

		fbAlmTrigTm(IN := NOT p_bAlarmSig);

		IF fbAlmTrigTm.Q = TRUE THEN
			eStatus		:= Error;
			udiStatus	:= 10006;	//Motorized Puller Alarm Occur

			bCW			:= FALSE;
			bCCW		:= FALSE;
			bSpdBinBit0	:= FALSE;
			bSpdBinBit1	:= FALSE;
			bSpdBinBit2	:= FALSE;
			bSigOn		:= FALSE;
			bBrake		:= FALSE;
			bAlmRst		:= FALSE;

			p_eAct	:= MtrPshrActIdle;
			eStat	:= MtrPshrActIdle;
		END_IF

	END_IF

	//Reset Error
	IF (eStatus = Error) AND bRstErr THEN
		IF p_bAlarmSig = FALSE THEN
			bAlmRst			:= TRUE;
			fbAlmRstTm.IN	:= TRUE;
			fbAlmTrigTm(IN := FALSE);
		END_IF
	END_IF

	fbAlmRstTm;

	IF fbAlmRstTm.Q = TRUE THEN
		bAlmRst		:= FALSE;
		eStatus		:= Idle;
		udiStatus	:= 0;

		fbAlmRstTm.IN	:= FALSE;
	END_IF

END_ACTION
```

#### Act_InitGlobal.st
```iecst
(** 2019-04-09 **)
ACTION Act_InitGlobal:

	(* Always Change If Project Change *)

	//Pass Data To Link
	p_bLinkOpsRun ACCESS p_OpsRun;

	p_bLinkDISafetyRlySig ACCESS p_DISafetyRlySig;
	p_bLinkPullConvPullerExtCtrl ACCESS p_PullConvPullerExtCtrl;
	p_bLinkPullConvPullerRetCtrl ACCESS p_PullConvPullerRetCtrl;
	p_bLinkAlarmSig ACCESS p_DIMtrPullerAlmSig;

	//Pass Data To Internal Use
	p_udiRstErr ACCESS p_RstErrReset;
	p_bPrep ACCESS p_NtParamProjMotorizedPullerPrep;
	p_bManual ACCESS p_UIMnlMod;
	p_bDir ACCESS p_NtParamMtrPshrDir;
	p_tExtTO ACCESS p_NtParamMtrPshrExtTO;
	p_tRetTO ACCESS p_NtParamMtrPshrRetTO;
	p_diExtSlowSpd ACCESS p_NtParamMtrPshrExtSlowSpd;
	p_diRetSlowSpd ACCESS p_NtParamMtrPshrRetSlowSpd;
	p_diExtNomSpd ACCESS p_NtParamMtrPshrExtNomSpd;
	p_diExtTorque ACCESS p_NtParamMtrPshrExtTorq;
	p_diStartTorque ACCESS p_NtParamMtrPshrStartTorq;
	p_sProgNm ACCESS p_NtParamMtrPshrProgNm;
	p_bNtSettingsLoadDone ACCESS p_StartupNtSettingsLoadDone;

	p_bExtSen ACCESS p_DIPullerExtRS;
	p_bRetSen ACCESS p_DIPullerRetRS;
	p_bExtSlowSen ACCESS p_DIPullerExtSlwSen;
	p_bRetSlowSen ACCESS p_DIPullerRetSlwSen;
//	p_bAlarmSig ACCESS p_DIMtrPullerAlmSig;
	p_bTorqueSig ACCESS p_DIMtrPullerTorqueSig;

	(* Always Change If Project Change *)

END_ACTION
```

#### Act_Link.st
```iecst
(** 2019-03-29 **)
ACTION Act_Link:

	IF p_bLinkDISafetyRlySig = FALSE THEN
		bExtended	:= FALSE;
		bRetracted	:= FALSE;
	END_IF

	IF p_bManual = TRUE THEN
		p_diRetNomSpd ACCESS p_UIMnlMtrPshrRetSpd;
		p_diRetTorque ACCESS p_UIMnlMtrPshrRetTorq;
	ELSE
		p_diRetNomSpd ACCESS p_ProdRcpCurrRcp1MtrPshrExtSpd;
		p_diRetTorque ACCESS p_ProdRcpCurrRcp1MtrPshrExtTorq;
	END_IF

	IF p_bLinkDISafetyRlySig = TRUE THEN
		p_bAlarmSig := p_bLinkAlarmSig;
	ELSE
		p_bAlarmSig := TRUE;
	END_IF

END_ACTION
```
